KUKA KRL program: MyProgram_161().src

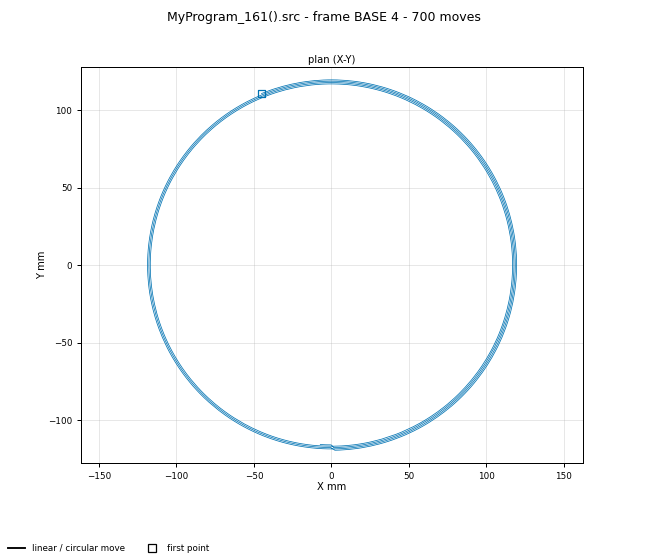
[picture p0: tool path of MyProgram_161().src in frame BASE 4, 700 of 700 moves have a stored position in this frame; points joined in program order, loops and branches not executed]
&ACCESS RVP
&REL 1
&PARAM TEMPLATE = C:\KRC\Roboter\Template\vorgabe
&PARAM EDITMASK = *
DEF MyProgram_161()
; ---- Setting reference (Base) ----
$BASE = BASE_DATA[4]

; --------------------------
; ---- Setting tool (TCP) ----
$TOOL = TOOL_DATA[3]
; --------------------------

$VEL.CP = VEL_APROX_PRINT
Startdeposition()
$VEL.CP = VEL_PRINT
LIN {X -45.1108,Y 110.7013,Z 123,A 107.6152,B 24.9409,C -1.7755,E1 24.9407,E2 338.4802} C_DIS
LIN {X -42.2928,Y 111.8083,Z 123,A 106.1798,B 24.9407,C -1.7782,E1 24.9444,E2 339.9124} C_DIS
LIN {X -39.6312,Y 112.7792,Z 123,A 104.7759,B 24.9407,C -1.7779,E1 24.9481,E2 341.3197} C_DIS
LIN {X -36.8224,Y 113.7272,Z 123,A 103.3582,B 24.9407,C -1.7798,E1 24.9519,E2 342.7356} C_DIS
LIN {X -33.9531,Y 114.6166,Z 123,A 101.9502,B 24.9404,C -1.7828,E1 24.9556,E2 344.1388} C_DIS
LIN {X -31.2205,Y 115.3909,Z 123,A 100.5452,B 24.9404,C -1.7823,E1 24.9594,E2 345.5472} C_DIS
LIN {X -28.2882,Y 116.1445,Z 123,A 99.1315,B 24.9403,C -1.7854,E1 24.9632,E2 346.9556} C_DIS
LIN {X -25.5209,Y 116.7838,Z 123,A 97.7268,B 24.9403,C -1.7847,E1 24.9671,E2 348.3636} C_DIS
LIN {X -22.5552,Y 117.3926,Z 123,A 96.3139,B 24.9401,C -1.7876,E1 24.9709,E2 349.7713} C_DIS
LIN {X -19.7599,Y 117.8954,Z 123,A 94.9099,B 24.9401,C -1.7867,E1 24.9748,E2 351.1788} C_DIS
LIN {X -16.7679,Y 118.358,Z 123,A 93.4767,B 24.9401,C -1.7885,E1 24.9787,E2 352.6089} C_DIS
LIN {X -13.8582,Y 118.7338,Z 123,A 92.0687,B 24.94,C -1.7893,E1 24.9826,E2 354.0162} C_DIS
LIN {X -11.0334,Y 119.0295,Z 123,A 90.6857,B 24.94,C -1.789,E1 24.9865,E2 355.4005} C_DIS
LIN {X -8.0155,Y 119.2708,Z 123,A 89.2737,B 24.9399,C -1.7914,E1 24.9904,E2 356.8075} C_DIS
LIN {X -5.1796,Y 119.4276,Z 123,A 87.8909,B 24.9399,C -1.7909,E1 24.9943,E2 358.1918} C_DIS
LIN {X -2.2472,Y 119.5187,Z 123,A 86.4636,B 24.9399,C -1.7903,E1 24.9982,E2 359.6205} C_DIS
LIN {X 0.6866,Y 119.5379,Z 123,A 85.0568,B 24.9399,C -1.7906,E1 25.0022,E2 361.0266} C_DIS
LIN {X 3.7137,Y 119.4821,Z 123,A 83.6459,B 24.9398,C -1.7926,E1 25.0061,E2 362.4326} C_DIS
LIN {X 6.6448,Y 119.355,Z 123,A 82.2396,B 24.9398,C -1.7926,E1 25.01,E2 363.8384} C_DIS
LIN {X 9.4785,Y 119.1635,Z 123,A 80.8376,B 24.9398,C -1.7907,E1 25.0139,E2 365.2441} C_DIS
LIN {X 12.4933,Y 118.8852,Z 123,A 79.4276,B 24.9398,C -1.7924,E1 25.0178,E2 366.6493} C_DIS
LIN {X 15.3142,Y 118.5548,Z 123,A 78.0264,B 24.9399,C -1.7903,E1 25.0217,E2 368.0544} C_DIS
LIN {X 18.219,Y 118.1433,Z 123,A 76.6411,B 24.9399,C -1.7909,E1 25.0256,E2 369.4371} C_DIS
LIN {X 21.1129,Y 117.6606,Z 123,A 75.236,B 24.9399,C -1.7904,E1 25.0294,E2 370.8418} C_DIS
LIN {X 23.9941,Y 117.107,Z 123,A 73.8109,B 24.94,C -1.7889,E1 25.0333,E2 372.2687} C_DIS
LIN {X 26.8608,Y 116.4829,Z 123,A 72.406,B 24.94,C -1.7882,E1 25.0372,E2 373.6733} C_DIS
LIN {X 29.7114,Y 115.7886,Z 123,A 71.022,B 24.94,C -1.7884,E1 25.0409,E2 375.0548} C_DIS
LIN {X 32.4883,Y 115.0404,Z 123,A 69.6114,B 24.9402,C -1.786,E1 25.0447,E2 376.4688} C_DIS
LIN {X 35.3571,Y 114.1913,Z 123,A 68.2138,B 24.9402,C -1.7866,E1 25.0484,E2 377.8625} C_DIS
LIN {X 38.1488,Y 113.2892,Z 123,A 66.8112,B 24.9402,C -1.7856,E1 25.0521,E2 379.2649} C_DIS
LIN {X 40.9176,Y 112.3188,Z 123,A 65.4066,B 24.9403,C -1.7844,E1 25.0558,E2 380.6695} C_DIS
LIN {X 43.6617,Y 111.2808,Z 123,A 64.0033,B 24.9404,C -1.7831,E1 25.0595,E2 382.0727} C_DIS
LIN {X 46.4659,Y 110.1394,Z 123,A 62.5554,B 24.9404,C -1.7817,E1 25.0632,E2 383.5205} C_DIS
LIN {X 49.0694,Y 109.0044,Z 123,A 61.1971,B 24.9406,C -1.7803,E1 25.0667,E2 384.8788} C_DIS
LIN {X 51.8142,Y 107.7268,Z 123,A 59.7701,B 24.9406,C -1.7797,E1 25.0703,E2 386.3037} C_DIS
LIN {X 54.4423,Y 106.4228,Z 123,A 58.3567,B 24.9408,C -1.7775,E1 25.0738,E2 387.7183} C_DIS
LIN {X 57.0377,Y 105.0546,Z 123,A 56.9656,B 24.9408,C -1.7763,E1 25.0773,E2 389.1084} C_DIS
LIN {X 59.5174,Y 103.6699,Z 123,A 55.5679,B 24.9411,C -1.7727,E1 25.0807,E2 390.5105} C_DIS
LIN {X 62.1238,Y 102.1294,Z 123,A 54.1416,B 24.9411,C -1.7716,E1 25.0841,E2 391.9348} C_DIS
LIN {X 64.6114,Y 100.574,Z 123,A 52.7403,B 24.9413,C -1.7697,E1 25.0874,E2 393.3363} C_DIS
LIN {X 67.0602,Y 98.9581,Z 123,A 51.339,B 24.9414,C -1.7676,E1 25.0906,E2 394.7378} C_DIS
LIN {X 69.3923,Y 97.337,Z 123,A 49.9623,B 24.9416,C -1.7645,E1 25.0938,E2 396.117} C_DIS
LIN {X 71.835,Y 95.5484,Z 123,A 48.5571,B 24.9416,C -1.7641,E1 25.0969,E2 397.5182} C_DIS
LIN {X 74.1583,Y 93.7567,Z 123,A 47.1362,B 24.9419,C -1.7608,E1 25.1001,E2 398.9416} C_DIS
LIN {X 76.3648,Y 91.9684,Z 123,A 45.7804,B 24.942,C -1.7584,E1 25.103,E2 400.2978} C_DIS
LIN {X 78.5988,Y 90.0666,Z 123,A 44.3601,B 24.9423,C -1.755,E1 25.106,E2 401.7207} C_DIS
LIN {X 80.8545,Y 88.0472,Z 123,A 42.903,B 24.9425,C -1.7518,E1 25.109,E2 403.1796} C_DIS
LIN {X 83.4853,Y 85.5599,Z 123,A 41.2079,B 24.9426,C -1.75,E1 25.1124,E2 404.8719} C_DIS
LIN {X 85.5599,Y 83.4853,Z 123,A 39.808,B 24.9428,C -1.7472,E1 25.1152,E2 406.2724} C_DIS
LIN {X 87.583,Y 81.3605,Z 123,A 38.4086,B 24.943,C -1.7444,E1 25.1179,E2 407.6724} C_DIS
LIN {X 89.5533,Y 79.1865,Z 123,A 37.0095,B 24.9432,C -1.7415,E1 25.1205,E2 409.0721} C_DIS
LIN {X 91.4697,Y 76.965,Z 123,A 35.61,B 24.9434,C -1.7385,E1 25.123,E2 410.4722} C_DIS
LIN {X 93.3309,Y 74.697,Z 123,A 34.2108,B 24.9436,C -1.7354,E1 25.1255,E2 411.8721} C_DIS
LIN {X 95.136,Y 72.384,Z 123,A 32.8122,B 24.9438,C -1.7323,E1 25.1279,E2 413.2714} C_DIS
LIN {X 96.8837,Y 70.0275,Z 123,A 31.4133,B 24.944,C -1.7292,E1 25.1302,E2 414.6711} C_DIS
LIN {X 98.5731,Y 67.6287,Z 123,A 30.015,B 24.9442,C -1.7259,E1 25.1324,E2 416.0702} C_DIS
LIN {X 100.2031,Y 65.1893,Z 123,A 28.6165,B 24.9444,C -1.7226,E1 25.1345,E2 417.4695} C_DIS
LIN {X 101.7728,Y 62.7105,Z 123,A 27.05,B 24.9451,C -1.7112,E1 25.1369,E2 419.055} C_DIS
LIN {X 103.6232,Y 59.5987,Z 123,A 25.4724,B 24.9449,C -1.7141,E1 25.1391,E2 420.6176} C_DIS
LIN {X 105.0546,Y 57.0377,Z 123,A 24.0949,B 24.9451,C -1.7116,E1 25.1409,E2 421.9939} C_DIS
LIN {X 106.4654,Y 54.3589,Z 123,A 22.6522,B 24.9453,C -1.7079,E1 25.1428,E2 423.4376} C_DIS
LIN {X 107.7674,Y 51.7297,Z 123,A 21.2746,B 24.9455,C -1.7053,E1 25.1445,E2 424.8139} C_DIS
LIN {X 108.9659,Y 49.1548,Z 123,A 19.9014,B 24.9458,C -1.7008,E1 25.1461,E2 426.1903} C_DIS
LIN {X 110.1758,Y 46.3795,Z 123,A 18.4795,B 24.946,C -1.698,E1 25.1477,E2 427.611} C_DIS
LIN {X 111.2808,Y 43.6617,Z 123,A 17.082,B 24.9462,C -1.6943,E1 25.1491,E2 429.0096} C_DIS
LIN {X 112.3188,Y 40.9176,Z 123,A 15.6647,B 24.9465,C -1.6895,E1 25.1505,E2 430.4301} C_DIS
LIN {X 113.2892,Y 38.1488,Z 123,A 14.2673,B 24.9467,C -1.6857,E1 25.1518,E2 431.8287} C_DIS
LIN {X 114.1913,Y 35.3571,Z 123,A 12.887,B 24.9469,C -1.6827,E1 25.1529,E2 433.2083} C_DIS
LIN {X 114.999,Y 32.6342,Z 123,A 11.5179,B 24.9472,C -1.6781,E1 25.154,E2 434.5804} C_DIS
LIN {X 115.7886,Y 29.7114,Z 123,A 10.0763,B 24.9475,C -1.6741,E1 25.155,E2 436.0231} C_DIS
LIN {X 116.4618,Y 26.9521,Z 123,A 8.7038,B 24.9478,C -1.6693,E1 25.1559,E2 437.3991} C_DIS
LIN {X 117.107,Y 23.9941,Z 123,A 7.2825,B 24.948,C -1.6662,E1 25.1567,E2 438.8194} C_DIS
LIN {X 117.644,Y 21.2052,Z 123,A 5.9302,B 24.9482,C -1.6623,E1 25.1574,E2 440.1729} C_DIS
LIN {X 118.1433,Y 18.219,Z 123,A 4.4949,B 24.9485,C -1.6584,E1 25.1581,E2 441.609} C_DIS
LIN {X 118.5548,Y 15.3142,Z 123,A 3.0925,B 24.9487,C -1.6541,E1 25.1586,E2 443.0133} C_DIS
LIN {X 118.8949,Y 12.4001,Z 123,A 1.7158,B 24.9489,C -1.651,E1 25.159,E2 444.3891} C_DIS
LIN {X 119.1635,Y 9.4785,Z 123,A 0.2992,B 24.9492,C -1.6459,E1 25.1594,E2 445.8092} C_DIS
LIN {X 119.355,Y 6.6448,Z 123,A -1.0527,B 24.9495,C -1.642,E1 25.1596,E2 447.1625} C_DIS
LIN {X 119.4821,Y 3.7137,Z 123,A -2.4491,B 24.9497,C -1.6379,E1 25.1597,E2 448.5602} C_DIS
LIN {X 119.5394,Y 0.5421,Z 123,A -4.0376,B 24.9502,C -1.6296,E1 25.1597,E2 450.1588} C_DIS
LIN {X 119.4821,Y -3.7137,Z 123,A -5.9849,B 24.9504,C -1.6274,E1 25.1597,E2 452.0996} C_DIS
LIN {X 119.355,Y -6.6448,Z 123,A -7.3614,B 24.9506,C -1.6243,E1 25.1595,E2 453.4752} C_DIS
LIN {X 119.1635,Y -9.4785,Z 123,A -8.7536,B 24.9509,C -1.6183,E1 25.1592,E2 454.8733} C_DIS
LIN {X 118.8852,Y -12.4933,Z 123,A -10.1543,B 24.9511,C -1.616,E1 25.1588,E2 456.2711} C_DIS
LIN {X 118.5548,Y -15.3142,Z 123,A -11.5463,B 24.9514,C -1.6101,E1 25.1583,E2 457.6689} C_DIS
LIN {X 118.1433,Y -18.219,Z 123,A -12.9076,B 24.9516,C -1.6077,E1 25.1578,E2 459.0278} C_DIS
LIN {X 117.644,Y -21.2052,Z 123,A -14.3438,B 24.9518,C -1.6037,E1 25.1571,E2 460.465} C_DIS
LIN {X 117.107,Y -23.9941,Z 123,A -15.7359,B 24.9522,C -1.5978,E1 25.1563,E2 461.8629} C_DIS
LIN {X 116.4618,Y -26.9521,Z 123,A -17.1368,B 24.9523,C -1.5955,E1 25.1555,E2 463.261} C_DIS
LIN {X 115.7886,Y -29.7114,Z 123,A -18.5091,B 24.9526,C -1.5906,E1 25.1546,E2 464.6369} C_DIS
LIN {X 115.0246,Y -32.544,Z 123,A -19.9056,B 24.9528,C -1.5866,E1 25.1535,E2 466.035} C_DIS
LIN {X 114.1913,Y -35.3571,Z 123,A -21.3024,B 24.9531,C -1.5826,E1 25.1524,E2 467.4333} C_DIS
LIN {X 113.2592,Y -38.2376,Z 123,A -22.744,B 24.9533,C -1.5784,E1 25.1511,E2 468.8765} C_DIS
LIN {X 112.2867,Y -41.0056,Z 123,A -24.1204,B 24.9535,C -1.5754,E1 25.1498,E2 470.2522} C_DIS
LIN {X 111.2466,Y -43.7489,Z 123,A -25.5378,B 24.9538,C -1.5705,E1 25.1484,E2 471.6733} C_DIS
LIN {X 110.1758,Y -46.3795,Z 123,A -26.91,B 24.9541,C -1.5657,E1 25.1469,E2 473.0492} C_DIS
LIN {X 108.9659,Y -49.1548,Z 123,A -28.3115,B 24.9541,C -1.5637,E1 25.1454,E2 474.448} C_DIS
LIN {X 107.7674,Y -51.7297,Z 123,A -29.6841,B 24.9545,C -1.559,E1 25.1437,E2 475.8243} C_DIS
LIN {X 106.4228,Y -54.4423,Z 123,A -31.1059,B 24.9546,C -1.556,E1 25.1419,E2 477.2455} C_DIS
LIN {X 105.0546,Y -57.0377,Z 123,A -32.5234,B 24.9549,C -1.5513,E1 25.1401,E2 478.6666} C_DIS
LIN {X 103.6699,Y -59.5174,Z 123,A -33.8961,B 24.9552,C -1.5467,E1 25.1382,E2 480.043} C_DIS
LIN {X 102.1294,Y -62.1238,Z 123,A -35.3184,B 24.9553,C -1.5439,E1 25.1361,E2 481.4647} C_DIS
LIN {X 100.6246,Y -64.5326,Z 123,A -36.671,B 24.9555,C -1.5404,E1 25.1341,E2 482.8187} C_DIS
LIN {X 99.0106,Y -66.9826,Z 123,A -38.0891,B 24.9558,C -1.5358,E1 25.1319,E2 484.2406} C_DIS
LIN {X 97.2825,Y -69.4685,Z 123,A -39.4913,B 24.9559,C -1.5341,E1 25.1297,E2 485.64} C_DIS
LIN {X 95.5484,Y -71.835,Z 123,A -40.9095,B 24.9562,C -1.5296,E1 25.1273,E2 487.0619} C_DIS
LIN {X 93.8148,Y -74.0848,Z 123,A -42.2628,B 24.9564,C -1.5263,E1 25.125,E2 488.4166} C_DIS
LIN {X 91.9684,Y -76.3648,Z 123,A -43.6614,B 24.9565,C -1.5229,E1 25.1225,E2 489.8167} C_DIS
LIN {X 90.0666,Y -78.5988,Z 123,A -45.0597,B 24.9567,C -1.5196,E1 25.1199,E2 491.2165} C_DIS
LIN {X 88.1106,Y -80.7855,Z 123,A -46.4584,B 24.9569,C -1.5164,E1 25.1173,E2 492.6167} C_DIS
LIN {X 86.1015,Y -82.9235,Z 123,A -47.8568,B 24.9571,C -1.5132,E1 25.1146,E2 494.0166} C_DIS
LIN {X 83.9738,Y -85.0774,Z 123,A -49.3004,B 24.9573,C -1.51,E1 25.1118,E2 495.4616} C_DIS
LIN {X 81.8606,Y -87.1126,Z 123,A -50.6992,B 24.9575,C -1.5069,E1 25.1089,E2 496.8618} C_DIS
LIN {X 79.6981,Y -89.0953,Z 123,A -52.0985,B 24.9576,C -1.5039,E1 25.106,E2 498.2625} C_DIS
LIN {X 77.4876,Y -91.0244,Z 123,A -53.4977,B 24.9578,C -1.501,E1 25.1031,E2 499.6632} C_DIS
LIN {X 75.2304,Y -92.8986,Z 123,A -54.8976,B 24.958,C -1.4982,E1 25.1,E2 501.0644} C_DIS
LIN {X 73.0022,Y -94.6597,Z 123,A -56.2524,B 24.9581,C -1.4955,E1 25.0971,E2 502.4206} C_DIS
LIN {X 70.5815,Y -96.4781,Z 123,A -57.6769,B 24.9582,C -1.4937,E1 25.0939,E2 503.8442} C_DIS
LIN {X 68.2695,Y -98.1277,Z 123,A -59.0726,B 24.9585,C -1.4892,E1 25.0907,E2 505.2456} C_DIS
LIN {X 65.7625,Y -99.8251,Z 123,A -60.4975,B 24.9585,C -1.4876,E1 25.0874,E2 506.6698} C_DIS
LIN {X 63.3724,Y -101.3593,Z 123,A -61.8529,B 24.9587,C -1.4852,E1 25.0842,E2 508.0263} C_DIS
LIN {X 60.8658,Y -102.884,Z 123,A -63.2739,B 24.9589,C -1.4818,E1 25.0808,E2 509.4508} C_DIS
LIN {X 58.3226,Y -104.3468,Z 123,A -64.6543,B 24.9589,C -1.4805,E1 25.0774,E2 510.8303} C_DIS
LIN {X 55.6613,Y -105.7903,Z 123,A -66.0799,B 24.959,C -1.4792,E1 25.0739,E2 512.2549} C_DIS
LIN {X 53.0483,Y -107.1245,Z 123,A -67.5014,B 24.9592,C -1.4761,E1 25.0703,E2 513.6798} C_DIS
LIN {X 50.4034,Y -108.3941,Z 123,A -68.8826,B 24.9592,C -1.475,E1 25.0669,E2 515.06} C_DIS
LIN {X 47.814,Y -109.5609,Z 123,A -70.28,B 24.9594,C -1.4712,E1 25.0633,E2 516.463} C_DIS
LIN {X 45.1108,Y -110.7013,Z 123,A -71.6614,B 24.9594,C -1.4704,E1 25.0597,E2 517.8432} C_DIS
LIN {X 42.2928,Y -111.8083,Z 123,A -73.0884,B 24.9595,C -1.4695,E1 25.056,E2 519.2692} C_DIS
LIN {X 39.6246,Y -112.7815,Z 123,A -74.4658,B 24.9597,C -1.4669,E1 25.0524,E2 520.6498} C_DIS
LIN {X 36.7557,Y -113.7488,Z 123,A -75.9133,B 24.9597,C -1.4653,E1 25.0485,E2 522.0985} C_DIS
LIN {X 33.9531,Y -114.6166,Z 123,A -77.3161,B 24.9599,C -1.4638,E1 25.0448,E2 523.5023} C_DIS
LIN {X 31.1301,Y -115.4153,Z 123,A -78.719,B 24.9599,C -1.4624,E1 25.041,E2 524.9061} C_DIS
LIN {X 28.2882,Y -116.1445,Z 123,A -80.102,B 24.9599,C -1.4621,E1 25.0373,E2 526.288} C_DIS
LIN {X 25.5435,Y -116.7789,Z 123,A -81.4954,B 24.9601,C -1.4588,E1 25.0334,E2 527.6872} C_DIS
LIN {X 22.5552,Y -117.3926,Z 123,A -82.909,B 24.9601,C -1.4598,E1 25.0296,E2 529.0967} C_DIS
LIN {X 19.7599,Y -117.8954,Z 123,A -84.3083,B 24.9602,C -1.4569,E1 25.0257,E2 530.5013} C_DIS
LIN {X 16.8606,Y -118.3448,Z 123,A -85.7127,B 24.9602,C -1.456,E1 25.0218,E2 531.9066} C_DIS
LIN {X 13.8582,Y -118.7338,Z 123,A -87.1213,B 24.9602,C -1.4571,E1 25.0179,E2 533.3116} C_DIS
LIN {X 11.0334,Y -119.0295,Z 123,A -88.5214,B 24.9604,C -1.4545,E1 25.014,E2 534.7168} C_DIS
LIN {X 8.0155,Y -119.2708,Z 123,A -89.9308,B 24.9604,C -1.4558,E1 25.0101,E2 536.1226} C_DIS
LIN {X 5.1796,Y -119.4276,Z 123,A -91.3113,B 24.9604,C -1.4543,E1 25.0063,E2 537.506} C_DIS
LIN {X 2.2472,Y -119.5187,Z 123,A -92.7367,B 24.9604,C -1.453,E1 25.0023,E2 538.9343} C_DIS
LIN {X 2.2472,Y -119.5187,Z 123,A -92.7367,B 24.9604,C -1.453,E1 25.0023,E2 538.9343} C_DIS
Enddeposition()
LIN {X 0.8403,Y -118.6613,Z 123,A -93.1387,B 24.9589,C -1.4807,E1 25.0014,E2 539.2706} C_DIS
Startdeposition()
$VEL.CP = VEL_PRINT
LIN {X 3.568,Y -118.6138,Z 123,A -91.5072,B 24.9581,C -1.4955,E1 25.006,E2 537.6044} C_DIS
LIN {X 6.3304,Y -118.4986,Z 123,A -90.0662,B 24.9578,C -1.5009,E1 25.0101,E2 536.151} C_DIS
LIN {X 9.3518,Y -118.2984,Z 123,A -88.669,B 24.9579,C -1.4986,E1 25.0139,E2 534.76} C_DIS
LIN {X 12.4477,Y -118.0128,Z 123,A -87.1181,B 24.9577,C -1.5017,E1 25.0183,E2 533.2026} C_DIS
LIN {X 16.0833,Y -117.5741,Z 123,A -85.2772,B 24.9575,C -1.5063,E1 25.0234,E2 531.3525} C_DIS
LIN {X 19.1587,Y -117.1114,Z 123,A -83.8011,B 24.9575,C -1.5062,E1 25.0274,E2 529.878} C_DIS
LIN {X 22.7634,Y -116.4641,Z 123,A -82.1126,B 24.9576,C -1.5039,E1 25.0321,E2 528.1967} C_DIS
LIN {X 26.2974,Y -115.7177,Z 123,A -80.2031,B 24.9571,C -1.5133,E1 25.0373,E2 526.2676} C_DIS
LIN {X 30.2459,Y -114.7504,Z 123,A -78.2448,B 24.957,C -1.5151,E1 25.0426,E2 524.308} C_DIS
LIN {X 34.3472,Y -113.5896,Z 123,A -76.3796,B 24.9574,C -1.5084,E1 25.0476,E2 522.462} C_DIS
LIN {X 37.9373,Y -112.4398,Z 123,A -74.5478,B 24.9572,C -1.5112,E1 25.0524,E2 520.627} C_DIS
LIN {X 41.8516,Y -111.0425,Z 123,A -72.6129,B 24.9572,C -1.5105,E1 25.0575,E2 518.6978} C_DIS
LIN {X 44.8351,Y -109.8716,Z 123,A -71.2656,B 24.9577,C -1.5032,E1 25.0609,E2 517.3707} C_DIS
LIN {X 48.0778,Y -108.4941,Z 123,A -69.1377,B 24.9564,C -1.526,E1 25.0665,E2 515.1941} C_DIS
LIN {X 51.8732,Y -106.7305,Z 123,A -67.2015,B 24.9564,C -1.5252,E1 25.0714,E2 513.2647} C_DIS
LIN {X 54.5025,Y -105.4122,Z 123,A -65.9219,B 24.9567,C -1.5209,E1 25.0745,E2 511.9988} C_DIS
LIN {X 57.5334,Y -103.7882,Z 123,A -64.4111,B 24.9569,C -1.5167,E1 25.0782,E2 510.5022} C_DIS
LIN {X 60.7458,Y -101.9415,Z 123,A -62.3126,B 24.9559,C -1.5348,E1 25.0834,E2 508.3673} C_DIS
LIN {X 64.2424,Y -99.7742,Z 123,A -60.5651,B 24.9563,C -1.5272,E1 25.0874,E2 506.6433} C_DIS
LIN {X 66.9618,Y -97.9711,Z 123,A -58.7814,B 24.9555,C -1.5404,E1 25.0916,E2 504.8346} C_DIS
LIN {X 70.0306,Y -95.8002,Z 123,A -57.0352,B 24.9555,C -1.5409,E1 25.0956,E2 503.0933} C_DIS
LIN {X 72.2698,Y -94.1226,Z 123,A -55.5857,B 24.9551,C -1.5486,E1 25.0988,E2 501.6309} C_DIS
LIN {X 75.6214,Y -91.4519,Z 123,A -53.647,B 24.9551,C -1.5469,E1 25.103,E2 499.7035} C_DIS
LIN {X 78.0063,Y -89.4258,Z 123,A -52.0941,B 24.9548,C -1.5524,E1 25.1063,E2 498.1438} C_DIS
LIN {X 80.8523,Y -86.8632,Z 123,A -50.2887,B 24.9548,C -1.5547,E1 25.11,E2 496.3403} C_DIS
LIN {X 83.9344,Y -83.8896,Z 123,A -48.134,B 24.9542,C -1.564,E1 25.1143,E2 494.1727} C_DIS
LIN {X 86.5039,Y -81.2345,Z 123,A -46.4205,B 24.9542,C -1.5651,E1 25.1176,E2 492.464} C_DIS
LIN {X 89.1057,Y -78.3728,Z 123,A -44.6348,B 24.9541,C -1.5659,E1 25.1209,E2 490.6843} C_DIS
LIN {X 91.8225,Y -75.1726,Z 123,A -42.7295,B 24.9541,C -1.5654,E1 25.1243,E2 488.7891} C_DIS
LIN {X 93.9949,Y -72.4355,Z 123,A -40.9351,B 24.9535,C -1.5752,E1 25.1274,E2 486.9799} C_DIS
LIN {X 96.3055,Y -69.3358,Z 123,A -39.2307,B 24.9537,C -1.5724,E1 25.1302,E2 485.2902} C_DIS
LIN {X 97.8449,Y -67.1477,Z 123,A -37.7129,B 24.9528,C -1.5871,E1 25.1327,E2 483.7454} C_DIS
LIN {X 99.8504,Y -64.1236,Z 123,A -36.0471,B 24.9528,C -1.5879,E1 25.1352,E2 482.0859} C_DIS
LIN {X 101.8767,Y -60.8556,Z 123,A -33.7542,B 24.9511,C -1.6147,E1 25.1386,E2 479.7415} C_DIS
LIN {X 103.7503,Y -57.6013,Z 123,A -32.4215,B 24.9522,C -1.5965,E1 25.1403,E2 478.4588} C_DIS
LIN {X 105.6063,Y -54.1228,Z 123,A -30.6098,B 24.9522,C -1.5977,E1 25.1427,E2 476.6538} C_DIS
LIN {X 107.1718,Y -50.9548,Z 123,A -28.5541,B 24.9508,C -1.62,E1 25.1452,E2 474.5564} C_DIS
LIN {X 109.2059,Y -46.4346,Z 123,A -26.4194,B 24.9511,C -1.6147,E1 25.1476,E2 472.446} C_DIS
LIN {X 110.4389,Y -43.419,Z 123,A -24.7228,B 24.9505,C -1.6256,E1 25.1494,E2 470.7329} C_DIS
LIN {X 111.8916,Y -39.5258,Z 123,A -22.9232,B 24.9507,C -1.6218,E1 25.1511,E2 468.9524} C_DIS
LIN {X 112.8375,Y -36.7383,Z 123,A -21.5278,B 24.9505,C -1.625,E1 25.1523,E2 467.5573} C_DIS
LIN {X 113.7047,Y -33.9593,Z 123,A -20.1525,B 24.9503,C -1.628,E1 25.1534,E2 466.1828} C_DIS
LIN {X 115.0323,Y -29.1491,Z 123,A -17.5828,B 24.9494,C -1.6436,E1 25.1553,E2 463.5911} C_DIS
LIN {X 116.0903,Y -24.6062,Z 123,A -15.3629,B 24.949,C -1.6493,E1 25.1566,E2 461.3707} C_DIS
LIN {X 116.7749,Y -21.1086,Z 123,A -13.7239,B 24.949,C -1.6509,E1 25.1575,E2 459.7375} C_DIS
LIN {X 117.3581,Y -17.5881,Z 123,A -12.095,B 24.9489,C -1.6519,E1 25.1582,E2 458.1159} C_DIS
LIN {X 117.7904,Y -14.4139,Z 123,A -10.4153,B 24.9481,C -1.6635,E1 25.1588,E2 456.4188} C_DIS
LIN {X 118.189,Y -10.6484,Z 123,A -8.6694,B 24.9481,C -1.6654,E1 25.1592,E2 454.6787} C_DIS
LIN {X 118.4716,Y -6.8197,Z 123,A -6.95,B 24.9481,C -1.6649,E1 25.1596,E2 452.9706} C_DIS
LIN {X 118.5928,Y -4.2521,Z 123,A -5.5169,B 24.9472,C -1.6784,E1 25.1597,E2 451.5143} C_DIS
LIN {X 118.6648,Y -0.8532,Z 123,A -3.9904,B 24.9472,C -1.6781,E1 25.1597,E2 449.9975} C_DIS
LIN {X 118.6348,Y 2.8609,Z 123,A -2.079,B 24.9465,C -1.6897,E1 25.1597,E2 448.0701} C_DIS
LIN {X 118.4658,Y 6.9247,Z 123,A -0.1756,B 24.9463,C -1.6932,E1 25.1594,E2 446.1699} C_DIS
LIN {X 118.1787,Y 10.7594,Z 123,A 1.5977,B 24.9462,C -1.6951,E1 25.159,E2 444.4026} C_DIS
LIN {X 117.8128,Y 14.2221,Z 123,A 3.2926,B 24.9458,C -1.7012,E1 25.1585,E2 442.7034} C_DIS
LIN {X 117.3032,Y 17.943,Z 123,A 5.1196,B 24.9454,C -1.7077,E1 25.1577,E2 440.8719} C_DIS
LIN {X 116.757,Y 21.2084,Z 123,A 6.7564,B 24.9449,C -1.7146,E1 25.1569,E2 439.2282} C_DIS
LIN {X 115.963,Y 25.1904,Z 123,A 8.6213,B 24.9449,C -1.7161,E1 25.1559,E2 437.3706} C_DIS
LIN {X 115.1628,Y 28.6313,Z 123,A 10.3139,B 24.9445,C -1.7208,E1 25.1548,E2 435.6768} C_DIS
LIN {X 114.14,Y 32.4657,Z 123,A 12.2049,B 24.9442,C -1.7255,E1 25.1534,E2 433.7856} C_DIS
LIN {X 113.2868,Y 35.3285,Z 123,A 13.6922,B 24.9438,C -1.7321,E1 25.1522,E2 432.2911} C_DIS
LIN {X 111.7738,Y 39.8614,Z 123,A 16.0508,B 24.9432,C -1.7415,E1 25.15,E2 429.9236} C_DIS
LIN {X 110.3735,Y 43.5853,Z 123,A 17.9038,B 24.943,C -1.744,E1 25.1481,E2 428.0752} C_DIS
LIN {X 108.8389,Y 47.2871,Z 123,A 19.7725,B 24.9428,C -1.7464,E1 25.1461,E2 426.211} C_DIS
LIN {X 107.1274,Y 51.0473,Z 123,A 21.7364,B 24.9426,C -1.7506,E1 25.1438,E2 424.2477} C_DIS
LIN {X 105.683,Y 53.9728,Z 123,A 23.3597,B 24.9421,C -1.7574,E1 25.1418,E2 422.6171} C_DIS
LIN {X 103.9563,Y 57.2318,Z 123,A 25.1293,B 24.9418,C -1.7618,E1 25.1394,E2 420.8465} C_DIS
LIN {X 101.8609,Y 60.8822,Z 123,A 27.1368,B 24.9415,C -1.7661,E1 25.1366,E2 418.8391} C_DIS
LIN {X 99.6282,Y 64.4698,Z 123,A 29.5117,B 24.9401,C -1.7877,E1 25.1329,E2 416.4252} C_DIS
LIN {X 97.698,Y 67.3592,Z 123,A 30.8107,B 24.941,C -1.7737,E1 25.131,E2 415.1656} C_DIS
LIN {X 95.7064,Y 70.1587,Z 123,A 32.4717,B 24.9407,C -1.778,E1 25.1282,E2 413.5025} C_DIS
LIN {X 92.8931,Y 73.844,Z 123,A 34.6551,B 24.9406,C -1.7808,E1 25.1245,E2 411.3228} C_DIS
LIN {X 90.5915,Y 76.6504,Z 123,A 36.4669,B 24.9401,C -1.7878,E1 25.1213,E2 409.5027} C_DIS
LIN {X 88.222,Y 79.3657,Z 123,A 38.1497,B 24.9401,C -1.7891,E1 25.1181,E2 407.8244} C_DIS
LIN {X 86.1403,Y 81.621,Z 123,A 39.7127,B 24.9395,C -1.7963,E1 25.1151,E2 406.2512} C_DIS
LIN {X 83.4665,Y 84.3522,Z 123,A 41.4268,B 24.9397,C -1.7941,E1 25.1118,E2 404.5498} C_DIS
LIN {X 80.9953,Y 86.7288,Z 123,A 43.1037,B 24.9394,C -1.7986,E1 25.1084,E2 402.8691} C_DIS
LIN {X 78.2968,Y 89.1721,Z 123,A 44.9006,B 24.939,C -1.804,E1 25.1046,E2 401.0666} C_DIS
LIN {X 75.2968,Y 91.7216,Z 123,A 47.1563,B 24.9376,C -1.8245,E1 25.0997,E2 398.7711} C_DIS
LIN {X 72.6121,Y 93.8588,Z 123,A 48.3989,B 24.9387,C -1.8079,E1 25.0971,E2 397.5723} C_DIS
LIN {X 70.1192,Y 95.7353,Z 123,A 49.8625,B 24.9387,C -1.8086,E1 25.0938,E2 396.1124} C_DIS
LIN {X 67.1073,Y 97.8726,Z 123,A 51.8006,B 24.938,C -1.8189,E1 25.0893,E2 394.1565} C_DIS
LIN {X 63.8401,Y 100.0325,Z 123,A 53.6448,B 24.938,C -1.8197,E1 25.085,E2 392.3163} C_DIS
LIN {X 60.5156,Y 102.0776,Z 123,A 55.4665,B 24.938,C -1.8197,E1 25.0806,E2 390.5005} C_DIS
LIN {X 57.4252,Y 103.8486,Z 123,A 57.1131,B 24.938,C -1.8187,E1 25.0766,E2 388.8612} C_DIS
LIN {X 54.1329,Y 105.6011,Z 123,A 59.0128,B 24.9375,C -1.8257,E1 25.0719,E2 386.9501} C_DIS
LIN {X 50.5087,Y 107.3827,Z 123,A 60.9536,B 24.9374,C -1.8277,E1 25.067,E2 385.0097} C_DIS
LIN {X 47.092,Y 108.9239,Z 123,A 62.5909,B 24.9378,C -1.8217,E1 25.0629,E2 383.3906} C_DIS
LIN {X 43.3063,Y 110.4831,Z 123,A 64.6049,B 24.9375,C -1.8255,E1 25.0577,E2 381.3722} C_DIS
LIN {X 38.7532,Y 112.1627,Z 123,A 66.9613,B 24.9373,C -1.8282,E1 25.0515,E2 379.0142} C_DIS
LIN {X 35.4482,Y 113.2496,Z 123,A 68.6351,B 24.9373,C -1.8293,E1 25.047,E2 377.3409} C_DIS
LIN {X 32.2654,Y 114.1968,Z 123,A 70.4208,B 24.9366,C -1.8389,E1 25.0422,E2 375.5356} C_DIS
LIN {X 28.2947,Y 115.2449,Z 123,A 72.2938,B 24.9369,C -1.835,E1 25.0372,E2 373.6745} C_DIS
LIN {X 24.8705,Y 116.0327,Z 123,A 73.883,B 24.9372,C -1.831,E1 25.0329,E2 372.097} C_DIS
LIN {X 21.7671,Y 116.6559,Z 123,A 75.5858,B 24.9366,C -1.8396,E1 25.0281,E2 370.3758} C_DIS
LIN {X 18.1668,Y 117.2686,Z 123,A 77.1822,B 24.937,C -1.8326,E1 25.0238,E2 368.7976} C_DIS
LIN {X 14.7034,Y 117.7543,Z 123,A 79.048,B 24.9365,C -1.841,E1 25.0186,E2 366.9134} C_DIS
LIN {X 10.6101,Y 118.1925,Z 123,A 81.0293,B 24.9365,C -1.841,E1 25.0131,E2 364.9334} C_DIS
LIN {X 6.666,Y 118.4801,Z 123,A 82.8249,B 24.9368,C -1.8359,E1 25.0081,E2 363.1507} C_DIS
LIN {X 3.273,Y 118.6228,Z 123,A 84.5664,B 24.9365,C -1.8403,E1 25.0032,E2 361.399} C_DIS
LIN {X -0.6126,Y 118.6659,Z 123,A 86.3994,B 24.9367,C -1.838,E1 24.9981,E2 359.5716} C_DIS
LIN {X -4.78,Y 118.5715,Z 123,A 88.421,B 24.9367,C -1.8378,E1 24.9925,E2 357.5501} C_DIS
LIN {X -8.5099,Y 118.363,Z 123,A 90.2717,B 24.9366,C -1.8392,E1 24.9873,E2 355.6956} C_DIS
LIN {X -12.2772,Y 118.0306,Z 123,A 91.9961,B 24.937,C -1.8338,E1 24.9825,E2 353.9831} C_DIS
LIN {X -16.3173,Y 117.5408,Z 123,A 94.0323,B 24.9368,C -1.8357,E1 24.9769,E2 351.9409} C_DIS
LIN {X -19.9302,Y 116.9824,Z 123,A 95.866,B 24.9368,C -1.8375,E1 24.9718,E2 350.1012} C_DIS
LIN {X -23.7548,Y 116.2655,Z 123,A 97.4872,B 24.9376,C -1.8246,E1 24.9675,E2 348.5089} C_DIS
LIN {X -27.3337,Y 115.4783,Z 123,A 99.4961,B 24.937,C -1.8335,E1 24.9619,E2 346.4762} C_DIS
LIN {X -33.8153,Y 113.7475,Z 123,A 102.6319,B 24.9375,C -1.8255,E1 24.9535,E2 343.3545} C_DIS
LIN {X -37.4397,Y 112.6076,Z 123,A 104.9558,B 24.9362,C -1.8449,E1 24.9472,E2 340.9803} C_DIS
LIN {X -41.075,Y 111.3328,Z 123,A 106.314,B 24.9379,C -1.8204,E1 24.9438,E2 339.6777} C_DIS
LIN {X -44.5169,Y 110.0011,Z 123,A 108.1874,B 24.9378,C -1.8219,E1 24.9389,E2 337.7964} C_DIS
LIN {X -47.0157,Y 108.9572,Z 123,A 109.9156,B 24.9366,C -1.8384,E1 24.9344,E2 336.025} C_DIS
LIN {X -50.5358,Y 107.3701,Z 123,A 111.2506,B 24.9384,C -1.8124,E1 24.9311,E2 334.7486} C_DIS
LIN {X -54.3719,Y 105.479,Z 123,A 113.4918,B 24.9381,C -1.8166,E1 24.9255,E2 332.4912} C_DIS
LIN {X -57.8636,Y 103.6038,Z 123,A 115.3742,B 24.9385,C -1.812,E1 24.9209,E2 330.6146} C_DIS
LIN {X -61.4488,Y 101.5187,Z 123,A 117.3236,B 24.9389,C -1.806,E1 24.9162,E2 328.6735} C_DIS
LIN {X -64.6976,Y 99.4817,Z 123,A 119.3167,B 24.9387,C -1.8085,E1 24.9115,E2 326.668} C_DIS
LIN {X -67.7437,Y 97.4307,Z 123,A 121.0124,B 24.9392,C -1.8017,E1 24.9077,E2 324.9828} C_DIS
LIN {X -71.2074,Y 94.9287,Z 123,A 123.0333,B 24.9396,C -1.7955,E1 24.9031,E2 322.9694} C_DIS
LIN {X -74.0251,Y 92.7499,Z 123,A 124.7715,B 24.9398,C -1.7926,E1 24.8993,E2 321.2318} C_DIS
LIN {X -76.314,Y 90.8763,Z 123,A 127.1009,B 24.9373,C -1.8282,E1 24.8942,E2 318.8085} C_DIS
LIN {X -80.6887,Y 87.0154,Z 123,A 129.2856,B 24.9397,C -1.7943,E1 24.8898,E2 316.6959} C_DIS
LIN {X -84.0882,Y 83.7338,Z 123,A 131.3651,B 24.9406,C -1.7801,E1 24.8857,E2 314.6413} C_DIS
LIN {X -88.7322,Y 78.7958,Z 123,A 134.5079,B 24.9415,C -1.7663,E1 24.8798,E2 311.5177} C_DIS
LIN {X -90.908,Y 76.2759,Z 123,A 136.2636,B 24.9414,C -1.7684,E1 24.8766,E2 309.749} C_DIS
LIN {X -93.1264,Y 73.5487,Z 123,A 137.9275,B 24.9418,C -1.7624,E1 24.8737,E2 308.0914} C_DIS
LIN {X -95.3822,Y 70.6015,Z 123,A 139.735,B 24.9421,C -1.7582,E1 24.8706,E2 306.2854} C_DIS
LIN {X -97.9153,Y 67.0443,Z 123,A 141.9495,B 24.9421,C -1.7568,E1 24.8671,E2 304.0633} C_DIS
LIN {X -99.707,Y 64.3472,Z 123,A 143.4584,B 24.9426,C -1.7501,E1 24.8648,E2 302.5629} C_DIS
LIN {X -101.6048,Y 61.307,Z 123,A 145.1955,B 24.9429,C -1.7454,E1 24.8623,E2 300.828} C_DIS
LIN {X -104.3453,Y 56.5157,Z 123,A 147.7621,B 24.9437,C -1.7334,E1 24.8588,E2 298.2766} C_DIS
LIN {X -105.7147,Y 53.9107,Z 123,A 149.2598,B 24.9437,C -1.7324,E1 24.8568,E2 296.7733} C_DIS
LIN {X -107.2296,Y 50.8346,Z 123,A 151.0109,B 24.9438,C -1.7313,E1 24.8547,E2 295.0151} C_DIS
LIN {X -108.7314,Y 47.5337,Z 123,A 152.737,B 24.9442,C -1.725,E1 24.8528,E2 293.2948} C_DIS
LIN {X -110.115,Y 44.2373,Z 123,A 154.4807,B 24.9445,C -1.7204,E1 24.8509,E2 291.5524} C_DIS
LIN {X -111.4018,Y 40.8857,Z 123,A 156.2365,B 24.9448,C -1.7159,E1 24.8492,E2 289.7973} C_DIS
LIN {X -112.6694,Y 37.2563,Z 123,A 158.1947,B 24.9449,C -1.7143,E1 24.8474,E2 287.8317} C_DIS
LIN {X -113.8772,Y 33.378,Z 123,A 160.6633,B 24.9439,C -1.7295,E1 24.8454,E2 285.3125} C_DIS
LIN {X -115.0812,Y 28.9592,Z 123,A 162.1544,B 24.9463,C -1.692,E1 24.8445,E2 283.9022} C_DIS
LIN {X -115.783,Y 26.0144,Z 123,A 163.9698,B 24.9457,C -1.7022,E1 24.8433,E2 282.052} C_DIS
LIN {X -116.7079,Y 21.4812,Z 123,A 166.2892,B 24.9459,C -1.6985,E1 24.8421,E2 279.7275} C_DIS
LIN {X -117.4344,Y 17.0665,Z 123,A 168.184,B 24.9471,C -1.6804,E1 24.8413,E2 277.8647} C_DIS
LIN {X -117.8827,Y 13.6251,Z 123,A 169.8283,B 24.9475,C -1.6736,E1 24.8407,E2 276.2267} C_DIS
LIN {X -118.2249,Y 10.2588,Z 123,A 171.6603,B 24.9473,C -1.6766,E1 24.8403,E2 274.3766} C_DIS
LIN {X -118.4685,Y 6.8763,Z 123,A 173.0282,B 24.9484,C -1.6599,E1 24.84,E2 273.0402} C_DIS
LIN {X -118.6009,Y 3.9879,Z 123,A 174.5876,B 24.9482,C -1.6622,E1 24.8398,E2 271.466} C_DIS
LIN {X -118.6697,Y 0.0302,Z 123,A 176.4311,B 24.9488,C -1.6531,E1 24.8398,E2 269.6331} C_DIS
LIN {X -118.6228,Y -3.2751,Z 123,A 178.1293,B 24.9488,C -1.6522,E1 24.8398,E2 267.9268} C_DIS
LIN {X -118.4679,Y -6.8865,Z 123,A 179.9627,B 24.949,C -1.6503,E1 24.8402,E2 266.0869} C_DIS
LIN {X -118.12,Y -11.3958,Z 123,A -177.8494,B 24.9494,C -1.6434,E1 24.8407,E2 263.9023} C_DIS
LIN {X -117.71,Y -15.0452,Z 123,A -176.1867,B 24.95,C -1.6331,E1 24.8412,E2 262.2543} C_DIS
LIN {X -117.2277,Y -18.4314,Z 123,A -174.1422,B 24.9493,C -1.6444,E1 24.8421,E2 260.1706} C_DIS
LIN {X -116.6418,Y -21.8407,Z 123,A -172.7871,B 24.9505,C -1.6258,E1 24.8428,E2 258.8519} C_DIS
LIN {X -116.0075,Y -24.986,Z 123,A -171.2582,B 24.9508,C -1.6201,E1 24.8437,E2 257.3276} C_DIS
LIN {X -115.0773,Y -28.9743,Z 123,A -168.9948,B 24.9505,C -1.626,E1 24.8452,E2 255.0368} C_DIS
LIN {X -113.8111,Y -33.6006,Z 123,A -166.8915,B 24.9514,C -1.6099,E1 24.8468,E2 252.9597} C_DIS
LIN {X -112.5478,Y -37.6169,Z 123,A -164.8479,B 24.9518,C -1.6042,E1 24.8485,E2 250.9181} C_DIS
LIN {X -111.2963,Y -41.1751,Z 123,A -163.0532,B 24.9522,C -1.5976,E1 24.8502,E2 249.1289} C_DIS
LIN {X -109.9757,Y -44.5793,Z 123,A -161.4567,B 24.9529,C -1.5853,E1 24.8518,E2 247.5526} C_DIS
LIN {X -109.0658,Y -46.765,Z 123,A -159.0276,B 24.9498,C -1.6371,E1 24.8548,E2 244.9867} C_DIS
LIN {X -106.2314,Y -52.8856,Z 123,A -157.0403,B 24.9536,C -1.5733,E1 24.857,E2 243.1408} C_DIS
LIN {X -104.5419,Y -56.1532,Z 123,A -155.0348,B 24.9533,C -1.5781,E1 24.8596,E2 241.1131} C_DIS
LIN {X -102.7866,Y -59.3036,Z 123,A -153.3015,B 24.9536,C -1.573,E1 24.862,E2 239.3829} C_DIS
LIN {X -100.65,Y -62.8611,Z 123,A -151.2797,B 24.9539,C -1.5684,E1 24.8649,E2 237.3617} C_DIS
LIN {X -98.1843,Y -66.647,Z 123,A -149.1011,B 24.9542,C -1.5627,E1 24.8683,E2 235.1859} C_DIS
LIN {X -95.9505,Y -69.8253,Z 123,A -147.2409,B 24.9546,C -1.5573,E1 24.8713,E2 233.3295} C_DIS
LIN {X -93.9641,Y -72.4756,Z 123,A -145.5834,B 24.9546,C -1.5558,E1 24.8741,E2 231.6674} C_DIS
LIN {X -91.3228,Y -75.7766,Z 123,A -143.5888,B 24.955,C -1.549,E1 24.8776,E2 229.6799} C_DIS
LIN {X -89.3656,Y -78.0752,Z 123,A -142.0797,B 24.9551,C -1.5478,E1 24.8804,E2 228.1668} C_DIS
LIN {X -86.784,Y -80.9366,Z 123,A -140.2985,B 24.9556,C -1.5401,E1 24.8837,E2 226.3959} C_DIS
LIN {X -84.5281,Y -83.2885,Z 123,A -138.6429,B 24.9556,C -1.5403,E1 24.8869,E2 224.7329} C_DIS
LIN {X -82.0131,Y -85.7673,Z 123,A -136.9685,B 24.9558,C -1.5353,E1 24.8903,E2 223.0632} C_DIS
LIN {X -79.1069,Y -88.4536,Z 123,A -135.0474,B 24.956,C -1.5319,E1 24.8942,E2 221.1425} C_DIS
LIN {X -72.692,Y -93.7973,Z 123,A -130.7542,B 24.9558,C -1.5357,E1 24.9036,E2 216.8241} C_DIS
LIN {X -68.8768,Y -96.6331,Z 123,A -128.6627,B 24.9566,C -1.5227,E1 24.9083,E2 214.7561} C_DIS
LIN {X -65.6237,Y -98.8717,Z 123,A -126.7121,B 24.9566,C -1.5215,E1 24.9128,E2 212.8018} C_DIS
LIN {X -62.6042,Y -100.8105,Z 123,A -125.148,B 24.9572,C -1.5114,E1 24.9164,E2 211.2568} C_DIS
LIN {X -59.601,Y -102.6157,Z 123,A -123.2811,B 24.9569,C -1.5167,E1 24.9209,E2 209.3718} C_DIS
LIN {X -56.7991,Y -104.1915,Z 123,A -121.8024,B 24.9572,C -1.5113,E1 24.9245,E2 207.9016} C_DIS
LIN {X -53.2609,Y -106.0453,Z 123,A -119.8719,B 24.9573,C -1.5089,E1 24.9293,E2 205.9716} C_DIS
LIN {X -50.3162,Y -107.4723,Z 123,A -118.2885,B 24.9574,C -1.5072,E1 24.9333,E2 204.3882} C_DIS
LIN {X -46.6737,Y -109.1049,Z 123,A -116.4167,B 24.9577,C -1.5025,E1 24.9381,E2 202.523} C_DIS
LIN {X -43.0533,Y -110.5825,Z 123,A -114.3058,B 24.9572,C -1.5106,E1 24.9436,E2 200.3882} C_DIS
LIN {X -38.8811,Y -112.1178,Z 123,A -112.2344,B 24.9575,C -1.5054,E1 24.949,E2 198.3252} C_DIS
LIN {X -35.191,Y -113.3294,Z 123,A -110.3918,B 24.9577,C -1.5025,E1 24.9539,E2 196.4862} C_DIS
LIN {X -31.747,Y -114.3437,Z 123,A -108.6363,B 24.9577,C -1.5022,E1 24.9587,E2 194.7284} C_DIS
LIN {X -28.2929,Y -115.2454,Z 123,A -106.9226,B 24.9578,C -1.5008,E1 24.9633,E2 193.0155} C_DIS
LIN {X -24.303,Y -116.153,Z 123,A -104.8782,B 24.9577,C -1.503,E1 24.9689,E2 190.9634} C_DIS
LIN {X -21.02,Y -116.7909,Z 123,A -103.3427,B 24.9579,C -1.4988,E1 24.9731,E2 189.4363} C_DIS
LIN {X -17.2733,Y -117.405,Z 123,A -101.4176,B 24.9577,C -1.5025,E1 24.9784,E2 187.5008} C_DIS
LIN {X -13.1626,Y -117.9369,Z 123,A -99.4005,B 24.9577,C -1.5029,E1 24.984,E2 185.4814} C_DIS
LIN {X -9.4918,Y -118.2872,Z 123,A -97.6849,B 24.9579,C -1.4999,E1 24.9888,E2 183.7722} C_DIS
LIN {X -5.5897,Y -118.5367,Z 123,A -95.7597,B 24.9578,C -1.5017,E1 24.9942,E2 181.8422} C_DIS
LIN {X -2.34,Y -118.6444,Z 123,A -94.201,B 24.9578,C -1.5014,E1 24.9985,E2 180.2839} C_DIS
LIN {X 0.8403,Y -118.6613,Z 123,A -93.1372,B 24.959,C -1.4801,E1 25.0014,E2 179.2706} C_DIS
Enddeposition()
LIN {X 0.8403,Y -118.6613,Z 123,A -93.1372,B 24.959,C -1.4801,E1 25.0014,E2 179.2706} C_DIS
Startdeposition()
$VEL.CP = VEL_PRINT
LIN {X -0.4666,Y -117.7943,Z 123,A -94.1503,B 24.959,C -1.4781,E1 24.9985,E2 180.2884} C_DIS
LIN {X -3.8504,Y -117.7323,Z 123,A -95.7663,B 24.959,C -1.4792,E1 24.994,E2 181.902} C_DIS
LIN {X -7.6369,Y -117.5476,Z 123,A -97.6463,B 24.9591,C -1.4775,E1 24.9887,E2 183.7866} C_DIS
LIN {X -11.0815,Y -117.2729,Z 123,A -99.2563,B 24.9589,C -1.4807,E1 24.9843,E2 185.3897} C_DIS
LIN {X -14.5655,Y -116.8924,Z 123,A -101.1038,B 24.9593,C -1.4746,E1 24.9791,E2 187.2529} C_DIS
LIN {X -18.0187,Y -116.4087,Z 123,A -102.7303,B 24.9591,C -1.4781,E1 24.9746,E2 188.8723} C_DIS
LIN {X -21.714,Y -115.7777,Z 123,A -104.6205,B 24.9591,C -1.4758,E1 24.9694,E2 190.7701} C_DIS
LIN {X -26.9934,Y -114.6615,Z 123,A -107.051,B 24.9587,C -1.4856,E1 24.9629,E2 193.1803} C_DIS
LIN {X -29.648,Y -114.0034,Z 123,A -108.4285,B 24.9587,C -1.4843,E1 24.9591,E2 194.5629} C_DIS
LIN {X -32.7363,Y -113.1565,Z 123,A -110.2444,B 24.9593,C -1.4739,E1 24.9542,E2 196.4062} C_DIS
LIN {X -36.6715,Y -111.9421,Z 123,A -112.3376,B 24.9594,C -1.4716,E1 24.9486,E2 198.5088} C_DIS
LIN {X -41.461,Y -110.2575,Z 123,A -114.5566,B 24.9587,C -1.4847,E1 24.9428,E2 200.701} C_DIS
LIN {X -44.7579,Y -108.9611,Z 123,A -116.1776,B 24.9584,C -1.4909,E1 24.9386,E2 202.3109} C_DIS
LIN {X -46.9661,Y -108.0271,Z 123,A -117.3218,B 24.9582,C -1.4932,E1 24.9357,E2 203.4524} C_DIS
LIN {X -49.2832,Y -106.9908,Z 123,A -118.7386,B 24.9586,C -1.4866,E1 24.9321,E2 204.8883} C_DIS
LIN {X -52.5513,Y -105.4234,Z 123,A -120.8848,B 24.9594,C -1.4722,E1 24.9266,E2 207.0743} C_DIS
LIN {X -55.8631,Y -103.7067,Z 123,A -122.0355,B 24.9577,C -1.5033,E1 24.9239,E2 208.1543} C_DIS
LIN {X -61.3157,Y -100.5786,Z 123,A -125.3013,B 24.9579,C -1.4987,E1 24.916,E2 211.4409} C_DIS
LIN {X -64.4928,Y -98.5724,Z 123,A -127.1896,B 24.9579,C -1.4989,E1 24.9115,E2 213.3347} C_DIS
LIN {X -67.2893,Y -96.6841,Z 123,A -128.7861,B 24.9576,C -1.5036,E1 24.9079,E2 214.9255} C_DIS
LIN {X -70.1796,Y -94.6097,Z 123,A -130.484,B 24.9574,C -1.5079,E1 24.904,E2 216.619} C_DIS
LIN {X -74.0442,Y -91.6141,Z 123,A -133.6057,B 24.9589,C -1.4808,E1 24.8971,E2 219.8168} C_DIS
LIN {X -77.6808,Y -88.5518,Z 123,A -135.2085,B 24.957,C -1.5154,E1 24.8938,E2 221.3437} C_DIS
LIN {X -79.948,Y -86.511,Z 123,A -136.8138,B 24.9571,C -1.5132,E1 24.8905,E2 222.9605} C_DIS
LIN {X -83.1771,Y -83.4119,Z 123,A -138.7934,B 24.9564,C -1.5262,E1 24.8866,E2 224.9176} C_DIS
LIN {X -85.9849,Y -80.5128,Z 123,A -140.8844,B 24.9564,C -1.5251,E1 24.8825,E2 227.0202} C_DIS
LIN {X -89.4631,Y -76.6296,Z 123,A -143.4923,B 24.9563,C -1.5278,E1 24.8777,E2 229.6332} C_DIS
LIN {X -91.7145,Y -73.9203,Z 123,A -145.1523,B 24.9559,C -1.5342,E1 24.8748,E2 231.2858} C_DIS
LIN {X -94.719,Y -70.0304,Z 123,A -147.4449,B 24.9553,C -1.5441,E1 24.8709,E2 233.5656} C_DIS
LIN {X -96.4821,Y -67.5799,Z 123,A -149.0983,B 24.9556,C -1.5401,E1 24.8682,E2 235.2368} C_DIS
LIN {X -98.3992,Y -64.7555,Z 123,A -150.7707,B 24.9553,C -1.5439,E1 24.8656,E2 236.9085} C_DIS
LIN {X -100.6045,Y -61.2733,Z 123,A -152.7479,B 24.955,C -1.5504,E1 24.8627,E2 238.8804} C_DIS
LIN {X -102.2625,Y -58.4645,Z 123,A -154.3955,B 24.9549,C -1.5521,E1 24.8604,E2 240.5324} C_DIS
LIN {X -104.5247,Y -54.3199,Z 123,A -156.5789,B 24.9542,C -1.5632,E1 24.8575,E2 242.7011} C_DIS
LIN {X -105.9178,Y -51.5484,Z 123,A -158.8679,B 24.9558,C -1.5353,E1 24.8546,E2 245.0689} C_DIS
LIN {X -107.9451,Y -47.1542,Z 123,A -160.6797,B 24.9541,C -1.5643,E1 24.8526,E2 246.8214} C_DIS
LIN {X -109.4417,Y -43.5713,Z 123,A -162.5191,B 24.9537,C -1.5719,E1 24.8507,E2 248.653} C_DIS
LIN {X -110.8182,Y -39.9397,Z 123,A -164.2962,B 24.9531,C -1.5822,E1 24.849,E2 250.4157} C_DIS
LIN {X -111.9954,Y -36.5068,Z 123,A -166.0989,B 24.9529,C -1.5859,E1 24.8474,E2 252.2196} C_DIS
LIN {X -113.0057,Y -33.2481,Z 123,A -167.7542,B 24.9526,C -1.5912,E1 24.846,E2 253.8719} C_DIS
LIN {X -114.8917,Y -25.9969,Z 123,A -171.9199,B 24.9532,C -1.5811,E1 24.8432,E2 258.0861} C_DIS
LIN {X -115.6569,Y -22.3416,Z 123,A -173.5825,B 24.9524,C -1.5932,E1 24.8423,E2 259.7298} C_DIS
LIN {X -116.7386,Y -15.7523,Z 123,A -176.4506,B 24.9509,C -1.619,E1 24.8411,E2 262.5532} C_DIS
LIN {X -117.1247,Y -12.5515,Z 123,A -178.5773,B 24.952,C -1.6013,E1 24.8405,E2 264.7351} C_DIS
LIN {X -117.4689,Y -8.7792,Z 123,A -179.9733,B 24.9505,C -1.6254,E1 24.8402,E2 266.0819} C_DIS
LIN {X -117.6997,Y -4.7476,Z 123,A 178.0289,B 24.9502,C -1.6304,E1 24.8399,E2 268.0797} C_DIS
LIN {X -117.7928,Y -0.7925,Z 123,A 176.0802,B 24.9499,C -1.6357,E1 24.8398,E2 270.0277} C_DIS
LIN {X -117.7619,Y 2.8789,Z 123,A 174.0943,B 24.95,C -1.6333,E1 24.8398,E2 272.0311} C_DIS
LIN {X -117.53,Y 7.8966,Z 123,A 171.864,B 24.949,C -1.65,E1 24.8402,E2 274.2351} C_DIS
LIN {X -117.2383,Y 11.456,Z 123,A 169.9937,B 24.949,C -1.6502,E1 24.8407,E2 276.1161} C_DIS
LIN {X -116.8257,Y 15.0807,Z 123,A 168.2293,B 24.9486,C -1.6564,E1 24.8413,E2 277.8763} C_DIS
LIN {X -116.0352,Y 20.2932,Z 123,A 165.6806,B 24.948,C -1.6654,E1 24.8424,E2 280.4188} C_DIS
LIN {X -114.3912,Y 28.1131,Z 123,A 162.2698,B 24.946,C -1.6974,E1 24.8444,E2 283.7732} C_DIS
LIN {X -113.1377,Y 32.8029,Z 123,A 159.4857,B 24.9466,C -1.6875,E1 24.8464,E2 286.5971} C_DIS
LIN {X -112.3419,Y 35.4298,Z 123,A 157.794,B 24.9473,C -1.6772,E1 24.8479,E2 288.3231} C_DIS
LIN {X -111.0553,Y 39.2743,Z 123,A 156.157,B 24.946,C -1.6971,E1 24.8493,E2 289.922} C_DIS
LIN {X -110.0868,Y 41.9119,Z 123,A 154.7825,B 24.9458,C -1.7011,E1 24.8506,E2 291.2948} C_DIS
LIN {X -108.8898,Y 44.9331,Z 123,A 153.0911,B 24.9458,C -1.7014,E1 24.8524,E2 292.9948} C_DIS
LIN {X -107.422,Y 48.334,Z 123,A 151.2849,B 24.9454,C -1.7068,E1 24.8545,E2 294.7983} C_DIS
LIN {X -106.0505,Y 51.2742,Z 123,A 149.7892,B 24.9449,C -1.7149,E1 24.8562,E2 296.2827} C_DIS
LIN {X -104.7984,Y 53.7865,Z 123,A 148.4175,B 24.9446,C -1.7187,E1 24.858,E2 297.6526} C_DIS
LIN {X -103.4661,Y 56.3067,Z 123,A 145.9703,B 24.9471,C -1.6797,E1 24.8614,E2 300.2058} C_DIS
LIN {X -100.3572,Y 61.68,Z 123,A 143.9866,B 24.9439,C -1.7306,E1 24.8641,E2 302.0785} C_DIS
LIN {X -98.587,Y 64.4706,Z 123,A 141.563,B 24.9457,C -1.7017,E1 24.8679,E2 304.5829} C_DIS
LIN {X -95.7571,Y 68.6024,Z 123,A 139.6771,B 24.9438,C -1.731,E1 24.8709,E2 306.4085} C_DIS
LIN {X -93.4735,Y 71.6829,Z 123,A 137.9365,B 24.9432,C -1.7412,E1 24.8738,E2 308.133} C_DIS
LIN {X -91.0545,Y 74.7342,Z 123,A 135.9174,B 24.9432,C -1.741,E1 24.8773,E2 310.162} C_DIS
LIN {X -88.4085,Y 77.8448,Z 123,A 134.0983,B 24.9424,C -1.7531,E1 24.8806,E2 311.9605} C_DIS
LIN {X -84.6418,Y 81.9237,Z 123,A 131.4181,B 24.9419,C -1.7607,E1 24.8857,E2 314.6343} C_DIS
LIN {X -82.5905,Y 83.9913,Z 123,A 129.8334,B 24.9421,C -1.7572,E1 24.8889,E2 316.2341} C_DIS
LIN {X -80.0668,Y 86.4019,Z 123,A 128.2531,B 24.9415,C -1.7661,E1 24.892,E2 317.7997} C_DIS
LIN {X -75.663,Y 90.283,Z 123,A 125.5174,B 24.9408,C -1.7776,E1 24.8978,E2 320.5187} C_DIS
LIN {X -72.6253,Y 92.7443,Z 123,A 123.251,B 24.9415,C -1.7665,E1 24.9028,E2 322.82} C_DIS
LIN {X -68.0224,Y 96.1709,Z 123,A 120.5775,B 24.9408,C -1.7772,E1 24.9088,E2 325.4773} C_DIS
LIN {X -64.7846,Y 98.38,Z 123,A 118.741,B 24.9404,C -1.784,E1 24.913,E2 327.3039} C_DIS
LIN {X -62.1178,Y 100.0857,Z 123,A 117.1626,B 24.9403,C -1.7853,E1 24.9168,E2 328.8843} C_DIS
LIN {X -57.7979,Y 102.6413,Z 123,A 114.9217,B 24.9394,C -1.7981,E1 24.9221,E2 331.1013} C_DIS
LIN {X -54.013,Y 104.6826,Z 123,A 112.3574,B 24.9405,C -1.7817,E1 24.9285,E2 333.7118} C_DIS
LIN {X -50.8787,Y 106.2405,Z 123,A 110.7839,B 24.94,C -1.7899,E1 24.9325,E2 335.27} C_DIS
LIN {X -46.8389,Y 108.0825,Z 123,A 108.6848,B 24.9396,C -1.7957,E1 24.9378,E2 337.3603} C_DIS
LIN {X -43.0997,Y 109.627,Z 123,A 106.8154,B 24.9391,C -1.8027,E1 24.9426,E2 339.2172} C_DIS
LIN {X -38.2273,Y 111.4209,Z 123,A 104.257,B 24.939,C -1.8045,E1 24.9493,E2 341.7764} C_DIS
LIN {X -34.27,Y 112.7003,Z 123,A 101.4967,B 24.9409,C -1.7754,E1 24.9569,E2 344.6106} C_DIS
LIN {X -29.4894,Y 114.0441,Z 123,A 100.0202,B 24.938,C -1.8181,E1 24.9606,E2 345.9881} C_DIS
LIN {X -24.3157,Y 115.2598,Z 123,A 97.3043,B 24.9383,C -1.8147,E1 24.968,E2 348.7154} C_DIS
LIN {X -21.6514,Y 115.7898,Z 123,A 95.779,B 24.9388,C -1.8069,E1 24.9723,E2 350.2609} C_DIS
LIN {X -18.0558,Y 116.403,Z 123,A 93.6896,B 24.9396,C -1.7946,E1 24.9781,E2 352.3814} C_DIS
LIN {X -14.3636,Y 116.9179,Z 123,A 92.3763,B 24.9381,C -1.8173,E1 24.9816,E2 353.6417} C_DIS
LIN {X -10.5807,Y 117.3191,Z 123,A 90.3859,B 24.9384,C -1.8122,E1 24.9872,E2 355.6453} C_DIS
LIN {X -6.5629,Y 117.612,Z 123,A 88.5101,B 24.9381,C -1.8167,E1 24.9924,E2 357.5112} C_DIS
LIN {X -3.3582,Y 117.7474,Z 123,A 86.9841,B 24.9381,C -1.8187,E1 24.9966,E2 359.0328} C_DIS
LIN {X -0.5385,Y 117.7939,Z 123,A 85.5386,B 24.9382,C -1.8157,E1 25.0007,E2 360.4853} C_DIS
LIN {X 3.406,Y 117.7459,Z 123,A 83.6256,B 24.9382,C -1.8163,E1 25.006,E2 362.3968} C_DIS
LIN {X 6.7566,Y 117.6013,Z 123,A 82.0565,B 24.938,C -1.8191,E1 25.0104,E2 363.9587} C_DIS
LIN {X 10.0504,Y 117.3673,Z 123,A 80.2832,B 24.9385,C -1.8115,E1 25.0153,E2 365.7489} C_DIS
LIN {X 13.7504,Y 116.9897,Z 123,A 78.6172,B 24.9381,C -1.8176,E1 25.0199,E2 367.3993} C_DIS
LIN {X 16.7875,Y 116.5928,Z 123,A 77.1304,B 24.9381,C -1.8174,E1 25.024,E2 368.8854} C_DIS
LIN {X 20.4335,Y 116.01,Z 123,A 74.8471,B 24.9396,C -1.7951,E1 25.0305,E2 371.2191} C_DIS
LIN {X 24.1227,Y 115.2994,Z 123,A 73.5385,B 24.9381,C -1.8173,E1 25.0339,E2 372.4735} C_DIS
LIN {X 27.1439,Y 114.6267,Z 123,A 71.9474,B 24.9384,C -1.8127,E1 25.0382,E2 374.0734} C_DIS
LIN {X 31.8934,Y 113.3954,Z 123,A 69.6285,B 24.9384,C -1.8142,E1 25.0445,E2 376.3851} C_DIS
LIN {X 36.2896,Y 112.0657,Z 123,A 67.4512,B 24.9383,C -1.815,E1 25.0503,E2 378.5565} C_DIS
LIN {X 39.0229,Y 111.1435,Z 123,A 65.913,B 24.9388,C -1.8077,E1 25.0544,E2 380.109} C_DIS
LIN {X 42.3632,Y 109.9158,Z 123,A 64.2836,B 24.9386,C -1.8106,E1 25.0586,E2 381.7281} C_DIS
LIN {X 45.1339,Y 108.8073,Z 123,A 62.8614,B 24.9386,C -1.8104,E1 25.0623,E2 383.1475} C_DIS
LIN {X 49.1888,Y 107.0348,Z 123,A 60.1577,B 24.9404,C -1.783,E1 25.0693,E2 385.9093} C_DIS
LIN {X 52.6183,Y 105.3902,Z 123,A 58.8204,B 24.939,C -1.8039,E1 25.0725,E2 387.1935} C_DIS
LIN {X 55.907,Y 103.6829,Z 123,A 56.7209,B 24.9401,C -1.7879,E1 25.0778,E2 389.3249} C_DIS
LIN {X 59.9406,Y 101.404,Z 123,A 54.7592,B 24.9394,C -1.798,E1 25.0825,E2 391.2569} C_DIS
LIN {X 62.8459,Y 99.6309,Z 123,A 53.0475,B 24.9398,C -1.7928,E1 25.0865,E2 392.9754} C_DIS
LIN {X 65.9322,Y 97.6146,Z 123,A 50.7033,B 24.9416,C -1.7646,E1 25.0921,E2 395.3782} C_DIS
LIN {X 69.5671,Y 95.0583,Z 123,A 48.044,B 24.9434,C -1.7382,E1 25.0982,E2 398.0906} C_DIS
LIN {X 74.9244,Y 90.8967,Z 123,A 45.7771,B 24.9407,C -1.7792,E1 25.1029,E2 400.2521} C_DIS
LIN {X 77.7859,Y 88.46,Z 123,A 44.0195,B 24.9407,C -1.7788,E1 25.1066,E2 402.0037} C_DIS
LIN {X 80.6558,Y 85.8505,Z 123,A 42.1901,B 24.9407,C -1.7776,E1 25.1103,E2 403.8284} C_DIS
LIN {X 82.8947,Y 83.6908,Z 123,A 40.6523,B 24.9411,C -1.7732,E1 25.1134,E2 405.3702} C_DIS
LIN {X 86.2454,Y 80.2359,Z 123,A 38.4051,B 24.9411,C -1.7724,E1 25.1177,E2 407.6096} C_DIS
LIN {X 89.1055,Y 77.0468,Z 123,A 36.2006,B 24.9418,C -1.7619,E1 25.1218,E2 409.8289} C_DIS
LIN {X 91.5326,Y 74.1448,Z 123,A 33.8195,B 24.9438,C -1.7323,E1 25.1262,E2 412.269} C_DIS
LIN {X 94.2842,Y 70.6129,Z 123,A 30.9617,B 24.9461,C -1.6955,E1 25.131,E2 415.2} C_DIS
LIN {X 98.681,Y 64.3281,Z 123,A 28.631,B 24.9425,C -1.751,E1 25.1344,E2 417.3881} C_DIS
LIN {X 100.0502,Y 62.1746,Z 123,A 27.3248,B 24.943,C -1.7446,E1 25.1364,E2 418.7027} C_DIS
LIN {X 102.8403,Y 57.4415,Z 123,A 25.0241,B 24.9423,C -1.755,E1 25.1396,E2 420.9671} C_DIS
LIN {X 104.1181,Y 55.092,Z 123,A 23.3623,B 24.9436,C -1.7342,E1 25.1418,E2 422.6692} C_DIS
LIN {X 105.6744,Y 52.0448,Z 123,A 21.387,B 24.9449,C -1.7148,E1 25.1443,E2 424.6797} C_DIS
LIN {X 107.0948,Y 49.0599,Z 123,A 20.176,B 24.944,C -1.729,E1 25.1457,E2 425.8508} C_DIS
LIN {X 108.583,Y 45.6661,Z 123,A 18.3322,B 24.9444,C -1.7218,E1 25.1478,E2 427.7015} C_DIS
LIN {X 110.0398,Y 42.036,Z 123,A 16.3935,B 24.9449,C -1.7144,E1 25.1497,E2 429.6468} C_DIS
LIN {X 111.307,Y 38.5568,Z 123,A 14.2127,B 24.9464,C -1.691,E1 25.1518,E2 431.8707} C_DIS
LIN {X 112.4366,Y 35.1246,Z 123,A 13.1562,B 24.9446,C -1.719,E1 25.1526,E2 432.855} C_DIS
LIN {X 114.0312,Y 29.5397,Z 123,A 10.361,B 24.9451,C -1.7117,E1 25.1548,E2 435.6514} C_DIS
LIN {X 114.9007,Y 25.9581,Z 123,A 8.1766,B 24.9466,C -1.6873,E1 25.1562,E2 437.8807} C_DIS
LIN {X 115.87,Y 21.2116,Z 123,A 5.9437,B 24.9467,C -1.6858,E1 25.1574,E2 440.1042} C_DIS
LIN {X 116.423,Y 17.9262,Z 123,A 4.329,B 24.9471,C -1.6809,E1 25.1581,E2 441.7208} C_DIS
LIN {X 116.9788,Y 13.8434,Z 123,A 2.3572,B 24.9474,C -1.676,E1 25.1588,E2 443.6925} C_DIS
LIN {X 117.3279,Y 10.4854,Z 123,A 0.6325,B 24.9479,C -1.6667,E1 25.1593,E2 445.4289} C_DIS
LIN {X 117.6145,Y 6.519,Z 123,A -1.1761,B 24.9479,C -1.6665,E1 25.1596,E2 447.2273} C_DIS
LIN {X 117.7636,Y 2.788,Z 123,A -3.0951,B 24.9486,C -1.6556,E1 25.1598,E2 449.1605} C_DIS
LIN {X 117.7904,Y -1.1429,Z 123,A -4.9663,B 24.9489,C -1.6514,E1 25.1598,E2 451.0307} C_DIS
LIN {X 117.6866,Y -5.0528,Z 123,A -6.7627,B 24.9489,C -1.6503,E1 25.1596,E2 452.819} C_DIS
LIN {X 117.5039,Y -8.2831,Z 123,A -8.3804,B 24.9494,C -1.643,E1 25.1593,E2 454.4442} C_DIS
LIN {X 117.1693,Y -12.126,Z 123,A -10.1878,B 24.9496,C -1.6402,E1 25.1588,E2 456.2475} C_DIS
LIN {X 116.5131,Y -17.3433,Z 123,A -12.6622,B 24.9499,C -1.6358,E1 25.1579,E2 458.7177} C_DIS
LIN {X 115.9908,Y -20.5399,Z 123,A -14.3286,B 24.9504,C -1.6263,E1 25.1571,E2 460.3966} C_DIS
LIN {X 115.3033,Y -24.1035,Z 123,A -16.3053,B 24.9514,C -1.6104,E1 25.156,E2 462.3993} C_DIS
LIN {X 114.1738,Y -28.9847,Z 123,A -18.9948,B 24.9526,C -1.5905,E1 25.1542,E2 465.1201} C_DIS
LIN {X 113.0964,Y -32.9425,Z 123,A -20.3469,B 24.9511,C -1.6149,E1 25.1532,E2 466.407} C_DIS
LIN {X 112.3468,Y -35.4141,Z 123,A -21.8115,B 24.952,C -1.6009,E1 25.152,E2 467.8964} C_DIS
LIN {X 109.8822,Y -42.45,Z 123,A -25.2319,B 24.952,C -1.5993,E1 25.1488,E2 471.3012} C_DIS
LIN {X 108.539,Y -45.7706,Z 123,A -27.0738,B 24.9527,C -1.5891,E1 25.1468,E2 473.157} C_DIS
LIN {X 105.2549,Y -52.8913,Z 123,A -30.9483,B 24.9535,C -1.5746,E1 25.1422,E2 477.0449} C_DIS
LIN {X 100.8988,Y -60.789,Z 123,A -35.0219,B 24.9535,C -1.5766,E1 25.1367,E2 481.0926} C_DIS
LIN {X 98.6309,Y -64.404,Z 123,A -37.3396,B 24.9545,C -1.559,E1 25.1332,E2 483.44} C_DIS
LIN {X 95.4649,Y -69.0118,Z 123,A -39.9017,B 24.9545,C -1.5589,E1 25.1291,E2 485.9899} C_DIS
LIN {X 91.9725,Y -73.6018,Z 123,A -42.6944,B 24.9549,C -1.5518,E1 25.1243,E2 488.786} C_DIS
LIN {X 89.1105,Y -77.0411,Z 123,A -44.8011,B 24.955,C -1.5494,E1 25.1205,E2 490.8888} C_DIS
LIN {X 86.1942,Y -80.2902,Z 123,A -47.2065,B 24.9561,C -1.5305,E1 25.116,E2 493.3281} C_DIS
LIN {X 83.1105,Y -83.4776,Z 123,A -49.4675,B 24.9567,C -1.5203,E1 25.1115,E2 495.6037} C_DIS
LIN {X 79.8376,Y -86.6123,Z 123,A -51.3996,B 24.9563,C -1.5279,E1 25.1076,E2 497.51} C_DIS
LIN {X 77.0562,Y -89.0973,Z 123,A -53.3842,B 24.957,C -1.5156,E1 25.1034,E2 499.5157} C_DIS
LIN {X 73.4883,Y -92.0622,Z 123,A -55.9037,B 24.9579,C -1.4982,E1 25.0979,E2 502.0668} C_DIS
LIN {X 70.4075,Y -94.4385,Z 123,A -57.1779,B 24.9565,C -1.5232,E1 25.0952,E2 503.2773} C_DIS
LIN {X 68.3974,Y -95.9033,Z 123,A -59.131,B 24.9586,C -1.4858,E1 25.0905,E2 505.3118} C_DIS
LIN {X 64.6203,Y -98.4883,Z 123,A -60.5918,B 24.9569,C -1.5171,E1 25.0873,E2 506.6938} C_DIS
LIN {X 62.2682,Y -99.9918,Z 123,A -62.0622,B 24.9573,C -1.5092,E1 25.0838,E2 508.1781} C_DIS
LIN {X 55.7651,Y -103.7599,Z 123,A -65.2439,B 24.9564,C -1.5247,E1 25.0762,E2 511.3136} C_DIS
LIN {X 52.1875,Y -105.6037,Z 123,A -67.652,B 24.9578,C -1.5003,E1 25.0701,E2 513.7728} C_DIS
LIN {X 48.5279,Y -107.3346,Z 123,A -69.8515,B 24.9586,C -1.4865,E1 25.0645,E2 515.9994} C_DIS
LIN {X 45.4164,Y -108.6883,Z 123,A -71.3459,B 24.9583,C -1.4913,E1 25.0607,E2 517.4791} C_DIS
LIN {X 41.7604,Y -110.1441,Z 123,A -73.8619,B 24.96,C -1.4609,E1 25.0539,E2 520.0613} C_DIS
LIN {X 37.1983,Y -111.7683,Z 123,A -75.3582,B 24.958,C -1.4974,E1 25.0502,E2 521.4684} C_DIS
LIN {X 33.3771,Y -112.9675,Z 123,A -77.4528,B 24.9585,C -1.4883,E1 25.0446,E2 523.5807} C_DIS
LIN {X 30.0942,Y -113.8877,Z 123,A -79.6136,B 24.9599,C -1.4635,E1 25.0386,E2 525.7968} C_DIS
LIN {X 26.4029,Y -114.7979,Z 123,A -80.968,B 24.9587,C -1.4843,E1 25.0351,E2 527.1} C_DIS
LIN {X 22.2053,Y -115.6831,Z 123,A -82.9985,B 24.9587,C -1.4851,E1 25.0295,E2 529.1262} C_DIS
LIN {X 19.3271,Y -116.1987,Z 123,A -84.4993,B 24.9589,C -1.4804,E1 25.0254,E2 530.6366} C_DIS
LIN {X 15.3981,Y -116.7845,Z 123,A -86.4098,B 24.9589,C -1.48,E1 25.0201,E2 532.5463} C_DIS
LIN {X 12.1109,Y -117.1708,Z 123,A -87.9665,B 24.9589,C -1.4815,E1 25.0158,E2 534.0983} C_DIS
LIN {X 8.9955,Y -117.4517,Z 123,A -89.57,B 24.9591,C -1.477,E1 25.0113,E2 535.7117} C_DIS
LIN {X 5.101,Y -117.6845,Z 123,A -91.4254,B 24.9591,C -1.4782,E1 25.0061,E2 537.5636} C_DIS
LIN {X 1.386,Y -117.7887,Z 123,A -93.3148,B 24.9593,C -1.4739,E1 25.0008,E2 539.4628} C_DIS
LIN {X 1.386,Y -117.7887,Z 123,A -93.3148,B 24.9593,C -1.4739,E1 25.0008,E2 539.4628} C_DIS
Enddeposition()
LIN {X 0.8315,Y -116.919,Z 123,A -93.1621,B 24.9574,C -1.5082,E1 25.0015,E2 539.2288} C_DIS
Startdeposition()
$VEL.CP = VEL_PRINT
LIN {X 3.4644,Y -116.8713,Z 123,A -91.5406,B 24.9565,C -1.5236,E1 25.0061,E2 537.5712} C_DIS
LIN {X 6.4122,Y -116.7466,Z 123,A -90.0426,B 24.9563,C -1.5265,E1 25.0103,E2 536.0667} C_DIS
LIN {X 10.4211,Y -116.4577,Z 123,A -88.0238,B 24.9562,C -1.5298,E1 25.0159,E2 534.0413} C_DIS
LIN {X 14.4991,Y -116.0213,Z 123,A -86.055,B 24.9562,C -1.5291,E1 25.0214,E2 532.0756} C_DIS
LIN {X 18.0397,Y -115.5227,Z 123,A -84.332,B 24.9562,C -1.5291,E1 25.0261,E2 530.3543} C_DIS
LIN {X 21.6473,Y -114.9021,Z 123,A -82.031,B 24.9548,C -1.5539,E1 25.0326,E2 527.997} C_DIS
LIN {X 25.6259,Y -114.082,Z 123,A -80.6144,B 24.9562,C -1.5291,E1 25.0363,E2 526.6409} C_DIS
LIN {X 32.3491,Y -112.3595,Z 123,A -77.0635,B 24.9556,C -1.5396,E1 25.046,E2 523.0707} C_DIS
LIN {X 41.5371,Y -109.2958,Z 123,A -72.4111,B 24.9555,C -1.5412,E1 25.0582,E2 518.4237} C_DIS
LIN {X 45.0717,Y -107.8868,Z 123,A -70.5641,B 24.9554,C -1.5431,E1 25.063,E2 516.5766} C_DIS
LIN {X 52.8888,Y -104.2775,Z 123,A -66.5579,B 24.9556,C -1.5397,E1 25.0731,E2 512.5885} C_DIS
LIN {X 57.2216,Y -101.9639,Z 123,A -63.3888,B 24.9532,C -1.5799,E1 25.081,E2 509.3336} C_DIS
LIN {X 60.921,Y -99.7976,Z 123,A -61.8918,B 24.9547,C -1.5553,E1 25.0845,E2 507.8995} C_DIS
LIN {X 64.0492,Y -97.8199,Z 123,A -59.2231,B 24.9521,C -1.5995,E1 25.0909,E2 505.1351} C_DIS
LIN {X 68.6093,Y -94.6783,Z 123,A -57.4798,B 24.9545,C -1.5589,E1 25.0947,E2 503.4938} C_DIS
LIN {X 72.8847,Y -91.4273,Z 123,A -54.6366,B 24.9535,C -1.5746,E1 25.101,E2 500.624} C_DIS
LIN {X 75.1907,Y -89.5411,Z 123,A -52.9657,B 24.9528,C -1.588,E1 25.1046,E2 498.9279} C_DIS
LIN {X 79.3939,Y -85.8353,Z 123,A -50.0047,B 24.9517,C -1.6048,E1 25.1108,E2 495.9392} C_DIS
LIN {X 82.4012,Y -82.952,Z 123,A -48.4193,B 24.9528,C -1.5879,E1 25.1139,E2 494.4003} C_DIS
LIN {X 86.2414,Y -78.9514,Z 123,A -45.8035,B 24.9526,C -1.5899,E1 25.1189,E2 491.7911} C_DIS
LIN {X 90.3887,Y -74.1706,Z 123,A -42.6432,B 24.952,C -1.6009,E1 25.1246,E2 488.6194} C_DIS
LIN {X 94.2733,Y -69.1624,Z 123,A -39.701,B 24.952,C -1.6015,E1 25.1296,E2 485.6897} C_DIS
LIN {X 97.054,Y -65.2041,Z 123,A -37.2673,B 24.9514,C -1.6112,E1 25.1335,E2 483.2451} C_DIS
LIN {X 99.0714,Y -62.0948,Z 123,A -35.6268,B 24.9516,C -1.608,E1 25.1359,E2 481.6204} C_DIS
LIN {X 100.2932,Y -60.1043,Z 123,A -33.3666,B 24.948,C -1.6653,E1 25.1393,E2 479.2364} C_DIS
LIN {X 103.2998,Y -54.7736,Z 123,A -31.3615,B 24.9505,C -1.6259,E1 25.1418,E2 477.3348} C_DIS
LIN {X 104.5698,Y -52.309,Z 123,A -29.1577,B 24.9477,C -1.6711,E1 25.1447,E2 475.0363} C_DIS
LIN {X 106.9664,Y -47.2161,Z 123,A -27.2279,B 24.9497,C -1.6392,E1 25.1468,E2 473.1922} C_DIS
LIN {X 108.2483,Y -44.195,Z 123,A -25.7115,B 24.9497,C -1.6398,E1 25.1484,E2 471.6828} C_DIS
LIN {X 109.3204,Y -41.4722,Z 123,A -23.8139,B 24.9479,C -1.6667,E1 25.1503,E2 469.7321} C_DIS
LIN {X 110.575,Y -38.0002,Z 123,A -21.9159,B 24.9473,C -1.6768,E1 25.1521,E2 467.8211} C_DIS
LIN {X 111.8957,Y -33.9224,Z 123,A -20.4377,B 24.9488,C -1.6532,E1 25.1532,E2 466.407} C_DIS
LIN {X 113.4618,Y -28.2417,Z 123,A -17.6321,B 24.9485,C -1.6585,E1 25.1553,E2 463.6051} C_DIS
LIN {X 114.6884,Y -22.7573,Z 123,A -14.684,B 24.9473,C -1.6768,E1 25.157,E2 460.6311} C_DIS
LIN {X 115.309,Y -19.3577,Z 123,A -13.3003,B 24.9479,C -1.6673,E1 25.1577,E2 459.2777} C_DIS
LIN {X 116.2065,Y -12.9373,Z 123,A -9.8798,B 24.9465,C -1.6894,E1 25.159,E2 455.8254} C_DIS
LIN {X 116.5506,Y -9.3186,Z 123,A -8.1606,B 24.9463,C -1.6922,E1 25.1594,E2 454.1097} C_DIS
LIN {X 116.8015,Y -5.3272,Z 123,A -6.3277,B 24.9463,C -1.6925,E1 25.1597,E2 452.2871} C_DIS
LIN {X 116.9002,Y -2.2883,Z 123,A -4.7808,B 24.9458,C -1.7001,E1 25.1597,E2 450.7314} C_DIS
LIN {X 116.9171,Y 1.261,Z 123,A -2.9181,B 24.9451,C -1.7117,E1 25.1597,E2 448.8524} C_DIS
LIN {X 116.8243,Y 4.7976,Z 123,A -1.3764,B 24.9453,C -1.7081,E1 25.1597,E2 447.3283} C_DIS
LIN {X 116.6619,Y 7.8028,Z 123,A 0.1728,B 24.9448,C -1.7165,E1 25.1593,E2 445.7686} C_DIS
LIN {X 116.3933,Y 11.1181,Z 123,A 1.9155,B 24.9441,C -1.7272,E1 25.1589,E2 444.0109} C_DIS
LIN {X 115.9571,Y 14.9943,Z 123,A 3.678,B 24.9441,C -1.7262,E1 25.1583,E2 442.2613} C_DIS
LIN {X 115.4266,Y 18.6542,Z 123,A 5.5825,B 24.9435,C -1.7364,E1 25.1575,E2 440.344} C_DIS
LIN {X 114.2511,Y 24.8509,Z 123,A 8.5827,B 24.9431,C -1.7418,E1 25.1559,E2 437.3485} C_DIS
LIN {X 113.3476,Y 28.6946,Z 123,A 11.009,B 24.9412,C -1.7716,E1 25.1542,E2 434.8661} C_DIS
LIN {X 112.2831,Y 32.6115,Z 123,A 12.3193,B 24.9429,C -1.7449,E1 25.1533,E2 433.6259} C_DIS
LIN {X 110.6656,Y 37.7381,Z 123,A 15.1771,B 24.9417,C -1.7636,E1 25.1508,E2 430.7403} C_DIS
LIN {X 109.3812,Y 41.3117,Z 123,A 16.883,B 24.9418,C -1.7618,E1 25.1491,E2 429.0483} C_DIS
LIN {X 108.3591,Y 43.923,Z 123,A 18.2544,B 24.9416,C -1.7657,E1 25.1477,E2 427.6753} C_DIS
LIN {X 107.1835,Y 46.7182,Z 123,A 19.8007,B 24.9411,C -1.7729,E1 25.146,E2 426.1203} C_DIS
LIN {X 106.1547,Y 49.0122,Z 123,A 21.7903,B 24.9384,C -1.8129,E1 25.1436,E2 424.0472} C_DIS
LIN {X 103.7914,Y 53.84,Z 123,A 23.7249,B 24.9402,C -1.7866,E1 25.1412,E2 422.1849} C_DIS
LIN {X 100.4647,Y 59.8152,Z 123,A 27.0217,B 24.9397,C -1.7932,E1 25.1367,E2 418.8898} C_DIS
LIN {X 98.4898,Y 63.0133,Z 123,A 28.7427,B 24.9397,C -1.7923,E1 25.1341,E2 417.1795} C_DIS
LIN {X 94.4077,Y 68.9788,Z 123,A 32.2785,B 24.9392,C -1.801,E1 25.1285,E2 413.6405} C_DIS
LIN {X 92.2533,Y 71.8371,Z 123,A 34.4251,B 24.9376,C -1.8239,E1 25.1247,E2 411.45} C_DIS
LIN {X 90.1576,Y 74.4488,Z 123,A 35.7105,B 24.9385,C -1.811,E1 25.1225,E2 410.2009} C_DIS
LIN {X 87.7244,Y 77.3019,Z 123,A 37.6058,B 24.938,C -1.818,E1 25.119,E2 408.2977} C_DIS
LIN {X 83.6274,Y 81.7175,Z 123,A 40.5361,B 24.9377,C -1.8235,E1 25.1134,E2 405.3671} C_DIS
LIN {X 81.1861,Y 84.1409,Z 123,A 42.1196,B 24.9377,C -1.8224,E1 25.1103,E2 403.7929} C_DIS
LIN {X 78.6145,Y 86.5505,Z 123,A 43.8655,B 24.9374,C -1.8268,E1 25.1067,E2 402.0437} C_DIS
LIN {X 75.8308,Y 88.9976,Z 123,A 45.5936,B 24.9374,C -1.8263,E1 25.103,E2 400.3235} C_DIS
LIN {X 70.752,Y 93.0858,Z 123,A 48.8762,B 24.9368,C -1.8363,E1 25.0958,E2 397.0296} C_DIS
LIN {X 67.882,Y 95.1994,Z 123,A 51.0096,B 24.9353,C -1.8574,E1 25.0909,E2 394.8538} C_DIS
LIN {X 64.8012,Y 97.3241,Z 123,A 52.4079,B 24.9365,C -1.8401,E1 25.0878,E2 393.501} C_DIS
LIN {X 61.9608,Y 99.1552,Z 123,A 54.0326,B 24.9365,C -1.8413,E1 25.0839,E2 391.8788} C_DIS
LIN {X 58.967,Y 100.9661,Z 123,A 55.7008,B 24.9365,C -1.8417,E1 25.0799,E2 390.2147} C_DIS
LIN {X 54.2311,Y 103.5855,Z 123,A 58.3372,B 24.9362,C -1.8447,E1 25.0735,E2 387.579} C_DIS
LIN {X 48.2126,Y 106.5198,Z 123,A 61.6387,B 24.9359,C -1.8496,E1 25.0652,E2 384.2745} C_DIS
LIN {X 45.3563,Y 107.7669,Z 123,A 63.1271,B 24.9359,C -1.8495,E1 25.0614,E2 382.7899} C_DIS
LIN {X 42.057,Y 109.0989,Z 123,A 65.1734,B 24.9348,C -1.865,E1 25.056,E2 380.7114} C_DIS
LIN {X 37.6843,Y 110.6838,Z 123,A 67.282,B 24.9352,C -1.8593,E1 25.0504,E2 378.6205} C_DIS
LIN {X 34.7678,Y 111.6338,Z 123,A 69.0918,B 24.9341,C -1.8744,E1 25.0455,E2 376.7782} C_DIS
LIN {X 31.4795,Y 112.6059,Z 123,A 70.1028,B 24.9362,C -1.8453,E1 25.043,E2 375.8378} C_DIS
LIN {X 27.6353,Y 113.6098,Z 123,A 72.3652,B 24.9351,C -1.8607,E1 25.0368,E2 373.5425} C_DIS
LIN {X 24.525,Y 114.3222,Z 123,A 74.6786,B 24.9327,C -1.8954,E1 25.0303,E2 371.1498} C_DIS
LIN {X 19.4394,Y 115.2954,Z 123,A 76.3524,B 24.9353,C -1.8573,E1 25.0259,E2 369.5679} C_DIS
LIN {X 16.3292,Y 115.7768,Z 123,A 77.9803,B 24.935,C -1.8616,E1 25.0214,E2 367.9314} C_DIS
LIN {X 12.5363,Y 116.2491,Z 123,A 79.8609,B 24.935,C -1.8623,E1 25.0162,E2 366.0507} C_DIS
LIN {X 8.9444,Y 116.5805,Z 123,A 81.7165,B 24.9347,C -1.8663,E1 25.011,E2 364.1865} C_DIS
LIN {X 4.881,Y 116.8207,Z 123,A 83.626,B 24.935,C -1.8625,E1 25.0057,E2 362.2867} C_DIS
LIN {X 0.9299,Y 116.9191,Z 123,A 85.4812,B 24.9352,C -1.8586,E1 25.0005,E2 360.441} C_DIS
LIN {X -1.8257,Y 116.9088,Z 123,A 86.9647,B 24.9349,C -1.8642,E1 24.9964,E2 358.9443} C_DIS
LIN {X -5.4157,Y 116.7977,Z 123,A 88.7567,B 24.9348,C -1.865,E1 24.9914,E2 357.1499} C_DIS
LIN {X -9.1042,Y 116.5678,Z 123,A 90.4831,B 24.9351,C -1.8605,E1 24.9866,E2 355.4335} C_DIS
LIN {X -12.8139,Y 116.2201,Z 123,A 92.3787,B 24.935,C -1.8626,E1 24.9813,E2 353.5319} C_DIS
LIN {X -20.189,Y 115.1675,Z 123,A 95.9826,B 24.9353,C -1.858,E1 24.9714,E2 349.9358} C_DIS
LIN {X -23.5753,Y 114.5211,Z 123,A 98.6949,B 24.9322,C -1.9015,E1 24.9637,E2 347.117} C_DIS
LIN {X -29.8599,Y 113.0473,Z 123,A 101.7386,B 24.9328,C -1.893,E1 24.9555,E2 344.0891} C_DIS
LIN {X -35.4324,Y 111.4261,Z 123,A 103.7335,B 24.9357,C -1.8527,E1 24.9504,E2 342.1864} C_DIS
LIN {X -38.7027,Y 110.3313,Z 123,A 105.7443,B 24.9348,C -1.8644,E1 24.945,E2 340.1438} C_DIS
LIN {X -41.98,Y 109.1281,Z 123,A 107.2077,B 24.9357,C -1.8514,E1 24.9413,E2 338.7082} C_DIS
LIN {X -45.1886,Y 107.8375,Z 123,A 108.8207,B 24.9362,C -1.8455,E1 24.9371,E2 337.1056} C_DIS
LIN {X -50.2113,Y 105.5932,Z 123,A 111.6657,B 24.936,C -1.8478,E1 24.9299,E2 334.2482} C_DIS
LIN {X -54.2038,Y 103.5999,Z 123,A 113.6913,B 24.9367,C -1.8373,E1 24.9249,E2 332.2422} C_DIS
LIN {X -57.0647,Y 102.0515,Z 123,A 115.2902,B 24.9369,C -1.8347,E1 24.921,E2 330.6448} C_DIS
LIN {X -60.8325,Y 99.8514,Z 123,A 117.6527,B 24.9365,C -1.8403,E1 24.9153,E2 328.2617} C_DIS
LIN {X -64.5584,Y 97.4841,Z 123,A 119.5908,B 24.9375,C -1.8266,E1 24.9108,E2 326.3501} C_DIS
LIN {X -67.6964,Y 95.3318,Z 123,A 121.7649,B 24.9368,C -1.8359,E1 24.9058,E2 324.1463} C_DIS
LIN {X -71.0748,Y 92.8407,Z 123,A 123.6774,B 24.9375,C -1.8254,E1 24.9015,E2 322.2519} C_DIS
LIN {X -74.507,Y 90.1092,Z 123,A 125.4526,B 24.9389,C -1.8049,E1 24.8978,E2 320.5188} C_DIS
LIN {X -77.4107,Y 87.6273,Z 123,A 127.7988,B 24.9379,C -1.8205,E1 24.8927,E2 318.1261} C_DIS
LIN {X -81.2633,Y 84.0666,Z 123,A 130.1883,B 24.9388,C -1.8068,E1 24.8879,E2 315.7595} C_DIS
LIN {X -83.9444,Y 81.39,Z 123,A 132.3256,B 24.9383,C -1.814,E1 24.8837,E2 313.596} C_DIS
LIN {X -87.7863,Y 77.231,Z 123,A 135.1907,B 24.9385,C -1.8107,E1 24.8783,E2 310.7259} C_DIS
LIN {X -89.9217,Y 74.7327,Z 123,A 136.4398,B 24.9399,C -1.7914,E1 24.8762,E2 309.5172} C_DIS
LIN {X -92.2669,Y 71.8194,Z 123,A 138.1633,B 24.9405,C -1.7819,E1 24.8732,E2 307.8081} C_DIS
LIN {X -95.1938,Y 67.8899,Z 123,A 141.257,B 24.939,C -1.8042,E1 24.868,E2 304.6462} C_DIS
LIN {X -97.5623,Y 64.4398,Z 123,A 142.8977,B 24.9405,C -1.7813,E1 24.8655,E2 303.052} C_DIS
LIN {X -99.1235,Y 62.0115,Z 123,A 145.3034,B 24.938,C -1.8187,E1 24.8619,E2 300.5447} C_DIS
LIN {X -102.5294,Y 56.2039,Z 123,A 147.5469,B 24.9416,C -1.7648,E1 24.859,E2 298.418} C_DIS
LIN {X -103.9649,Y 53.5003,Z 123,A 148.9963,B 24.9421,C -1.7583,E1 24.8571,E2 296.9765} C_DIS
LIN {X -105.4967,Y 50.4122,Z 123,A 150.79,B 24.9421,C -1.7575,E1 24.8549,E2 295.1749} C_DIS
LIN {X -107.095,Y 46.9211,Z 123,A 152.6034,B 24.9427,C -1.7489,E1 24.8528,E2 293.372} C_DIS
LIN {X -108.3538,Y 43.9358,Z 123,A 154.2198,B 24.9429,C -1.7452,E1 24.8511,E2 291.7555} C_DIS
LIN {X -109.6725,Y 40.535,Z 123,A 155.8564,B 24.9437,C -1.7334,E1 24.8495,E2 290.1378} C_DIS
LIN {X -111.072,Y 36.527,Z 123,A 158.0613,B 24.9437,C -1.732,E1 24.8475,E2 287.9237} C_DIS
LIN {X -112.0452,Y 33.4183,Z 123,A 159.6029,B 24.9443,C -1.7247,E1 24.8463,E2 286.3907} C_DIS
LIN {X -113.196,Y 29.2847,Z 123,A 161.7543,B 24.9446,C -1.7199,E1 24.8447,E2 284.2381} C_DIS
LIN {X -114.5939,Y 23.2209,Z 123,A 164.9923,B 24.9446,C -1.7178,E1 24.8427,E2 280.9861} C_DIS
LIN {X -115.3863,Y 18.8957,Z 123,A 167.3265,B 24.9446,C -1.7182,E1 24.8416,E2 278.637} C_DIS
LIN {X -116.196,Y 13.0267,Z 123,A 170.1182,B 24.9456,C -1.7042,E1 24.8406,E2 275.8622} C_DIS
LIN {X -116.5819,Y 8.9274,Z 123,A 172.5202,B 24.945,C -1.7135,E1 24.8401,E2 273.4236} C_DIS
LIN {X -116.8126,Y 5.0701,Z 123,A 174.2862,B 24.9457,C -1.702,E1 24.8399,E2 271.6742} C_DIS
LIN {X -116.9101,Y 1.7529,Z 123,A 175.6713,B 24.9467,C -1.6867,E1 24.8398,E2 270.3172} C_DIS
LIN {X -116.905,Y -2.03,Z 123,A 177.4497,B 24.9473,C -1.6776,E1 24.8398,E2 268.5499} C_DIS
LIN {X -116.6738,Y -7.627,Z 123,A 179.941,B 24.9485,C -1.6582,E1 24.8402,E2 266.0898} C_DIS
LIN {X -116.1143,Y -13.7247,Z 123,A -176.903,B 24.9487,C -1.6549,E1 24.841,E2 262.9229} C_DIS
LIN {X -115.2878,Y -19.4848,Z 123,A -174.1686,B 24.9495,C -1.6409,E1 24.8421,E2 260.2056} C_DIS
LIN {X -114.1751,Y -25.1993,Z 123,A -170.989,B 24.9493,C -1.6453,E1 24.8439,E2 256.9966} C_DIS
LIN {X -112.6187,Y -31.4346,Z 123,A -167.8878,B 24.95,C -1.6335,E1 24.846,E2 253.9054} C_DIS
LIN {X -111.7422,Y -34.4182,Z 123,A -166.3247,B 24.9502,C -1.6305,E1 24.8473,E2 252.3405} C_DIS
LIN {X -110.7997,Y -37.3405,Z 123,A -164.8476,B 24.9505,C -1.6248,E1 24.8486,E2 250.8685} C_DIS
LIN {X -109.6958,Y -40.4709,Z 123,A -163.0563,B 24.9505,C -1.6268,E1 24.8503,E2 249.0624} C_DIS
LIN {X -108.2716,Y -44.1378,Z 123,A -160.8036,B 24.9499,C -1.6347,E1 24.8527,E2 246.7782} C_DIS
LIN {X -106.8208,Y -47.5447,Z 123,A -159.337,B 24.9511,C -1.6149,E1 24.8543,E2 245.3508} C_DIS
LIN {X -105.029,Y -51.3826,Z 123,A -157.2022,B 24.9513,C -1.6115,E1 24.8569,E2 243.2126} C_DIS
LIN {X -103.1443,Y -55.0689,Z 123,A -155.0822,B 24.9515,C -1.6096,E1 24.8596,E2 241.0856} C_DIS
LIN {X -101.0199,Y -58.8759,Z 123,A -152.9756,B 24.9519,C -1.6026,E1 24.8625,E2 238.9849} C_DIS
LIN {X -98.3007,Y -63.3078,Z 123,A -150.5559,B 24.9526,C -1.5905,E1 24.8661,E2 236.5817} C_DIS
LIN {X -96.0796,Y -66.6304,Z 123,A -148.55,B 24.9528,C -1.5874,E1 24.8692,E2 234.5731} C_DIS
LIN {X -93.4749,Y -70.2377,Z 123,A -145.8449,B 24.9518,C -1.6043,E1 24.8738,E2 231.8148} C_DIS
LIN {X -90.8838,Y -73.5597,Z 123,A -144.3512,B 24.9535,C -1.575,E1 24.8763,E2 230.3838} C_DIS
LIN {X -86.3081,Y -78.8787,Z 123,A -140.8761,B 24.9539,C -1.5686,E1 24.8827,E2 226.9083} C_DIS
LIN {X -83.9296,Y -81.4054,Z 123,A -139.0806,B 24.9539,C -1.5689,E1 24.8862,E2 225.1043} C_DIS
LIN {X -81.9732,Y -83.3748,Z 123,A -137.4399,B 24.9533,C -1.578,E1 24.8895,E2 223.435} C_DIS
LIN {X -79.5137,Y -85.7255,Z 123,A -136.0275,B 24.9542,C -1.5636,E1 24.8924,E2 222.0512} C_DIS
LIN {X -75.4792,Y -89.2971,Z 123,A -132.8227,B 24.9531,C -1.5828,E1 24.8993,E2 218.7881} C_DIS
LIN {X -71.8642,Y -92.2324,Z 123,A -131.0966,B 24.9547,C -1.5545,E1 24.9029,E2 217.123} C_DIS
LIN {X -69.0541,Y -94.3526,Z 123,A -129.4066,B 24.955,C -1.55,E1 24.9067,E2 215.4376} C_DIS
LIN {X -65.7927,Y -96.6555,Z 123,A -127.4618,B 24.9552,C -1.5462,E1 24.9112,E2 213.4952} C_DIS
LIN {X -62.7303,Y -98.6714,Z 123,A -125.5619,B 24.9552,C -1.5479,E1 24.9156,E2 211.5853} C_DIS
LIN {X -56.2721,Y -102.4924,Z 123,A -121.1302,B 24.9535,C -1.5758,E1 24.9266,E2 207.0743} C_DIS
LIN {X -51.287,Y -105.0763,Z 123,A -119.1263,B 24.9556,C -1.5393,E1 24.9314,E2 205.1517} C_DIS
LIN {X -48.0687,Y -106.5847,Z 123,A -117.7522,B 24.9566,C -1.5213,E1 24.9348,E2 203.8171} C_DIS
LIN {X -45.5847,Y -107.6706,Z 123,A -116.0658,B 24.9558,C -1.5355,E1 24.9392,E2 202.0929} C_DIS
LIN {X -41.4515,Y -109.3282,Z 123,A -113.97,B 24.9562,C -1.5296,E1 24.9446,E2 200.0066} C_DIS
LIN {X -38.001,Y -110.577,Z 123,A -112.243,B 24.9564,C -1.5249,E1 24.9491,E2 198.2875} C_DIS
LIN {X -34.4889,Y -111.7203,Z 123,A -109.9721,B 24.9553,C -1.544,E1 24.9553,E2 195.9672} C_DIS
LIN {X -31.1003,Y -112.7122,Z 123,A -108.528,B 24.9561,C -1.5301,E1 24.9591,E2 194.5539} C_DIS
LIN {X -27.5473,Y -113.6312,Z 123,A -106.1341,B 24.9547,C -1.5558,E1 24.9658,E2 192.0956} C_DIS
LIN {X -22.7729,Y -114.6854,Z 123,A -104.3276,B 24.9562,C -1.5282,E1 24.9706,E2 190.3524} C_DIS
LIN {X -19.2211,Y -115.3319,Z 123,A -102.6199,B 24.9564,C -1.5249,E1 24.9753,E2 188.6509} C_DIS
LIN {X -15.3694,Y -115.9085,Z 123,A -100.7955,B 24.9567,C -1.5207,E1 24.9803,E2 186.835} C_DIS
LIN {X -12.3921,Y -116.2642,Z 123,A -99.2804,B 24.9566,C -1.5226,E1 24.9845,E2 185.3146} C_DIS
LIN {X -9.046,Y -116.5724,Z 123,A -97.5918,B 24.9565,C -1.5244,E1 24.9892,E2 183.6208} C_DIS
LIN {X -5.0366,Y -116.814,Z 123,A -95.623,B 24.9565,C -1.5245,E1 24.9947,E2 181.6511} C_DIS
LIN {X -1.0179,Y -116.9185,Z 123,A -93.8482,B 24.9569,C -1.516,E1 24.9996,E2 179.8964} C_DIS
LIN {X 0.8315,Y -116.919,Z 123,A -93.158,B 24.9575,C -1.5065,E1 25.0015,E2 179.2288} C_DIS
Enddeposition()
LIN {X 0.8315,Y -116.919,Z 123,A -93.158,B 24.9575,C -1.5065,E1 25.0015,E2 179.2288} C_DIS
Startdeposition()
$VEL.CP = VEL_PRINT
LIN {X -0.2057,Y -116.0511,Z 123,A -94.1027,B 24.9577,C -1.5024,E1 24.9988,E2 180.1833} C_DIS
LIN {X -3.5279,Y -115.9965,Z 123,A -95.6984,B 24.9577,C -1.5041,E1 24.9944,E2 181.775} C_DIS
LIN {X -7.1835,Y -115.8294,Z 123,A -97.5393,B 24.9577,C -1.5025,E1 24.9892,E2 183.6204} C_DIS
Enddeposition()
END
